LIN {X -0.019,Y -439.634,Z 747.550,A 0.000,B 0.000,C 90.000,E1 134.960} C_DIS
LIN {X -0.236,Y -446.877,Z 747.546,A 0.000,B 0.000,C 90.000,E1 134.271} C_DIS
LIN {X -0.116,Y -458.331,Z 747.539,A 0.000,B 0.000,C 90.000,E1 133.095} C_DIS
LIN {X 0.017,Y -466.662,Z 747.535,A 0.000,B 0.000,C 90.000,E1 132.204} C_DIS
LIN {X 0.112,Y -474.907,Z 747.530,A 0.000,B 0.000,C 90.000,E1 131.310} C_DIS
LIN {X -0.249,Y -482.897,Z 747.525,A 0.000,B 0.000,C 90.000,E1 130.458} C_DIS
LIN {X 0.218,Y -489.352,Z 747.520,A 0.000,B 0.000,C 90.000,E1 129.644} C_DIS
LIN {X 0.055,Y -494.191,Z 747.517,A 0.000,B 0.000,C 90.000,E1 129.072} C_DIS
LIN {X 0.218,Y -496.646,Z 747.515,A 0.000,B 0.000,C 90.000,E1 128.749} C_DIS
LIN {X -0.083,Y -504.313,Z 747.510,A 0.000,B 0.000,C 90.000,E1 127.729} C_DIS
LIN {X 0.206,Y -509.388,Z 747.505,A 0.000,B 0.000,C 90.000,E1 126.950} C_DIS
LIN {X 0.138,Y -513.980,Z 747.501,A 0.000,B 0.000,C 90.000,E1 126.217} C_DIS
LIN {X 0.118,Y -517.480,Z 747.498,A 0.000,B 0.000,C 90.000,E1 125.644} C_DIS
LIN {X -0.310,Y -520.857,Z 747.495,A 0.000,B 0.000,C 90.000,E1 125.105} C_DIS
LIN {X 0.174,Y -526.566,Z 747.489,A 0.000,B 0.000,C 90.000,E1 123.913} C_DIS
LIN {X -0.212,Y -530.567,Z 747.484,A 0.000,B 0.000,C 90.000,E1 123.086} C_DIS
LIN {X 0.022,Y -535.010,Z 747.478,A 0.000,B 0.000,C 90.000,E1 122.054} C_DIS
LIN {X -0.107,Y -538.597,Z 747.473,A 0.000,B 0.000,C 90.000,E1 121.209} C_DIS
LIN {X 0.079,Y -541.957,Z 747.469,A 0.000,B 0.000,C 90.000,E1 120.335} C_DIS
LIN {X -0.181,Y -544.080,Z 747.465,A 0.000,B 0.000,C 90.000,E1 119.795} C_DIS
LIN {X -0.209,Y -547.156,Z 747.461,A 0.000,B 0.000,C 90.000,E1 118.949} C_DIS
LIN {X -0.201,Y -550.028,Z 747.456,A 0.000,B 0.000,C 90.000,E1 118.103} C_DIS
LIN {X -0.163,Y -552.767,Z 747.451,A 0.000,B 0.000,C 90.000,E1 117.257} C_DIS
LIN {X -0.099,Y -555.288,Z 747.447,A 0.000,B 0.000,C 90.000,E1 116.411} C_DIS
LIN {X -0.256,Y -557.387,Z 747.442,A 0.000,B 0.000,C 90.000,E1 115.591} C_DIS
LIN {X 0.120,Y -559.196,Z 747.437,A 0.000,B 0.000,C 90.000,E1 114.719} C_DIS
LIN {X -0.194,Y -561.181,Z 747.431,A 0.000,B 0.000,C 90.000,E1 113.643} C_DIS
LIN {X 0.028,Y -562.877,Z 747.425,A 0.000,B 0.000,C 90.000,E1 112.514} C_DIS
LIN {X -0.020,Y -565.156,Z 747.416,A 0.000,B 0.000,C 90.000,E1 110.865} C_DIS
LIN {X 0.045,Y -566.668,Z 747.410,A 0.000,B 0.000,C 90.000,E1 109.758} C_DIS
LIN {X -0.105,Y -568.686,Z 747.401,A 0.000,B 0.000,C 90.000,E1 108.127} C_DIS
LIN {X -0.220,Y -570.542,Z 747.392,A 0.000,B 0.000,C 90.000,E1 106.496} C_DIS
LIN {X 0.268,Y -572.608,Z 747.381,A 0.000,B 0.000,C 90.000,E1 104.537} C_DIS
LIN {X -0.093,Y -574.375,Z 747.372,A 0.000,B 0.000,C 90.000,E1 102.939} C_DIS
LIN {X -0.200,Y -575.877,Z 747.364,A 0.000,B 0.000,C 90.000,E1 101.591} C_DIS
LIN {X -0.178,Y -577.585,Z 747.355,A 0.000,B 0.000,C 90.000,E1 99.962} C_DIS
LIN {X 0.234,Y -578.955,Z 747.348,A 0.000,B 0.000,C 90.000,E1 98.568} C_DIS
LIN {X -0.199,Y -580.736,Z 747.337,A 0.000,B 0.000,C 90.000,E1 96.720} C_DIS
LIN {X 0.183,Y -581.859,Z 747.330,A 0.000,B 0.000,C 90.000,E1 95.334} C_DIS
LIN {X -0.057,Y -582.888,Z 747.322,A 0.000,B 0.000,C 90.000,E1 94.012} C_DIS
LIN {X -0.138,Y -584.060,Z 747.313,A 0.000,B 0.000,C 90.000,E1 92.407} C_DIS
LIN {X 0.026,Y -584.828,Z 747.307,A 0.000,B 0.000,C 90.000,E1 91.318} C_DIS
LIN {X 0.164,Y -585.782,Z 747.297,A 0.000,B 0.000,C 90.000,E1 89.427} C_DIS
LIN {X 0.146,Y -586.397,Z 747.288,A 0.000,B 0.000,C 90.000,E1 87.822} C_DIS
LIN {X 0.139,Y -586.904,Z 747.279,A 0.000,B 0.000,C 90.000,E1 86.216} C_DIS
LIN {X -0.197,Y -587.126,Z 747.273,A 0.000,B 0.000,C 90.000,E1 85.179} C_DIS
LIN {X -0.163,Y -587.343,Z 747.264,A 0.000,B 0.000,C 90.000,E1 83.571} C_DIS
LIN {X -0.247,Y -587.387,Z 747.257,A 0.000,B 0.000,C 90.000,E1 82.243} C_DIS
LIN {X -0.084,Y -587.316,Z 747.248,A 0.000,B 0.000,C 90.000,E1 80.622} C_DIS
LIN {X -0.083,Y -587.056,Z 747.240,A 0.000,B 0.000,C 90.000,E1 79.285} C_DIS
LIN {X 0.276,Y -586.543,Z 747.232,A 0.000,B 0.000,C 90.000,E1 77.645} C_DIS
LIN {X -0.195,Y -586.012,Z 747.224,A 0.000,B 0.000,C 90.000,E1 76.353} C_DIS
LIN {X -0.292,Y -585.221,Z 747.215,A 0.000,B 0.000,C 90.000,E1 74.755} C_DIS
LIN {X 0.082,Y -584.442,Z 747.208,A 0.000,B 0.000,C 90.000,E1 73.378} C_DIS
LIN {X 0.044,Y -583.756,Z 747.202,A 0.000,B 0.000,C 90.000,E1 72.308} C_DIS
LIN {X 0.228,Y -582.538,Z 747.193,A 0.000,B 0.000,C 90.000,E1 70.678} C_DIS
LIN {X -0.015,Y -581.674,Z 747.187,A 0.000,B 0.000,C 90.000,E1 69.625} C_DIS
LIN {X -0.071,Y -580.407,Z 747.179,A 0.000,B 0.000,C 90.000,E1 68.284} C_DIS
LIN {X 0.057,Y -578.988,Z 747.172,A 0.000,B 0.000,C 90.000,E1 66.922} C_DIS
LIN {X -0.374,Y -577.316,Z 747.164,A 0.000,B 0.000,C 90.000,E1 65.613} C_DIS
LIN {X 0.172,Y -575.385,Z 747.157,A 0.000,B 0.000,C 90.000,E1 64.204} C_DIS
LIN {X 0.074,Y -573.609,Z 747.151,A 0.000,B 0.000,C 90.000,E1 63.127} C_DIS
LIN {X 0.103,Y -572.094,Z 747.146,A 0.000,B 0.000,C 90.000,E1 62.308} C_DIS
LIN {X 0.043,Y -571.055,Z 747.143,A 0.000,B 0.000,C 90.000,E1 61.769} C_DIS
LIN {X 0.136,Y -568.559,Z 747.137,A 0.000,B 0.000,C 90.000,E1 60.667} C_DIS
LIN {X -0.120,Y -566.513,Z 747.133,A 0.000,B 0.000,C 90.000,E1 59.871} C_DIS
LIN {X 0.184,Y -563.488,Z 747.127,A 0.000,B 0.000,C 90.000,E1 58.742} C_DIS
LIN {X 0.172,Y -560.988,Z 747.122,A 0.000,B 0.000,C 90.000,E1 57.916} C_DIS
LIN {X -0.164,Y -558.261,Z 747.117,A 0.000,B 0.000,C 90.000,E1 57.120} C_DIS
LIN {X -0.152,Y -554.192,Z 747.111,A 0.000,B 0.000,C 90.000,E1 56.008} C_DIS
LIN {X -0.067,Y -550.147,Z 747.106,A 0.000,B 0.000,C 90.000,E1 55.022} C_DIS
LIN {X -0.086,Y -546.928,Z 747.102,A 0.000,B 0.000,C 90.000,E1 54.322} C_DIS
LIN {X -0.279,Y -542.565,Z 747.097,A 0.000,B 0.000,C 90.000,E1 53.497} C_DIS
LIN {X -0.072,Y -540.308,Z 747.095,A 0.000,B 0.000,C 90.000,E1 53.050} C_DIS
LIN {X -0.187,Y -536.083,Z 747.091,A 0.000,B 0.000,C 90.000,E1 52.351} C_DIS
LIN {X 0.152,Y -532.406,Z 747.088,A 0.000,B 0.000,C 90.000,E1 51.743} C_DIS
LIN {X 0.133,Y -528.356,Z 747.084,A 0.000,B 0.000,C 90.000,E1 51.170} C_DIS
LIN {X 0.082,Y -523.734,Z 747.081,A 0.000,B 0.000,C 90.000,E1 50.598} C_DIS
LIN {X -0.207,Y -519.937,Z 747.079,A 0.000,B 0.000,C 90.000,E1 50.194} C_DIS
LIN {X -0.127,Y -514.436,Z 747.076,A 0.000,B 0.000,C 90.000,E1 49.622} C_DIS
LIN {X -0.008,Y -508.929,Z 747.073,A 0.000,B 0.000,C 90.000,E1 49.094} C_DIS
LIN {X 0.013,Y -504.675,Z 747.071,A 0.000,B 0.000,C 90.000,E1 48.728} C_DIS
LIN {X -0.184,Y -497.064,Z 747.068,A 0.000,B 0.000,C 90.000,E1 48.162} C_DIS
LIN {X 0.042,Y -490.703,Z 747.065,A 0.000,B 0.000,C 90.000,E1 47.676} C_DIS
LIN {X 0.313,Y -485.892,Z 747.063,A 0.000,B 0.000,C 90.000,E1 47.310} C_DIS
LIN {X 0.124,Y -479.241,Z 747.061,A 0.000,B 0.000,C 90.000,E1 46.905} C_DIS
LIN {X 0.132,Y -464.679,Z 747.056,A 0.000,B 0.000,C 90.000,E1 45.972} C_DIS
LIN {X -0.056,Y -446.780,Z 747.049,A 0.000,B 0.000,C 90.000,E1 44.838} C_DIS
LIN {X -0.086,Y -424.493,Z 747.041,A 0.000,B 0.000,C 90.000,E1 43.299} C_DIS
LIN {X -0.037,Y -418.213,Z 747.038,A 0.000,B 0.000,C 90.000,E1 42.813} C_DIS
LIN {X 0.002,Y -413.026,Z 747.035,A 0.000,B 0.000,C 90.000,E1 42.366} C_DIS
LIN {X -0.027,Y -412.987,Z 747.035,A 0.000,B 0.000,C 90.000,E1 42.366} C_DIS
LIN {X -0.059,Y -405.949,Z 747.014,A 0.000,B 0.000,C 90.000,E1 38.543} C_DIS
LIN {X 0.058,Y -402.213,Z 747.004,A 0.000,B 0.000,C 90.000,E1 36.790} C_DIS
LIN {X -0.041,Y -401.945,Z 747.004,A 0.000,B 0.000,C 90.000,E1 36.629} C_DIS
LIN {X -0.022,Y -402.376,Z 746.987,A 0.000,B 0.000,C 90.000,E1 33.658} C_DIS
LIN {X -0.078,Y -403.741,Z 746.968,A 0.000,B 0.000,C 90.000,E1 30.178} C_DIS
LIN {X -0.117,Y -405.368,Z 746.950,A 0.000,B 0.000,C 90.000,E1 27.052} C_DIS
LIN {X 0.102,Y -406.865,Z 746.937,A 0.000,B 0.000,C 90.000,E1 24.591} C_DIS
LIN {X -0.051,Y -409.155,Z 746.921,A 0.000,B 0.000,C 90.000,E1 21.844} C_DIS
LIN {X -0.182,Y -412.799,Z 746.902,A 0.000,B 0.000,C 90.000,E1 18.417} C_DIS
LIN {X 0.068,Y -416.776,Z 746.885,A 0.000,B 0.000,C 90.000,E1 15.300} C_DIS
LIN {X -0.087,Y -420.303,Z 746.872,A 0.000,B 0.000,C 90.000,E1 12.939} C_DIS
LIN {X 0.010,Y -423.521,Z 746.861,A 0.000,B 0.000,C 90.000,E1 10.894} C_DIS
LIN {X 0.205,Y -427.248,Z 746.847,A 0.000,B 0.000,C 90.000,E1 8.511} C_DIS
LIN {X -0.099,Y -430.434,Z 746.836,A 0.000,B 0.000,C 90.000,E1 6.543} C_DIS
LIN {X 0.080,Y -434.348,Z 746.823,A 0.000,B 0.000,C 90.000,E1 4.188} C_DIS
LIN {X -0.182,Y -437.889,Z 746.812,A 0.000,B 0.000,C 90.000,E1 2.236} C_DIS
LIN {X 0.056,Y -441.622,Z 746.801,A 0.000,B 0.000,C 90.000,E1 0.229} C_DIS
LIN {X 0.214,Y -447.043,Z 746.786,A 0.000,B 0.000,C 90.000,E1 357.478} C_DIS
LIN {X 0.098,Y -450.544,Z 746.777,A 0.000,B 0.000,C 90.000,E1 355.869} C_DIS
LIN {X -0.037,Y -455.589,Z 746.765,A 0.000,B 0.000,C 90.000,E1 353.628} C_DIS
LIN {X 0.107,Y -459.211,Z 746.756,A 0.000,B 0.000,C 90.000,E1 352.008} C_DIS
LIN {X 0.078,Y -461.979,Z 746.749,A 0.000,B 0.000,C 90.000,E1 350.735} C_DIS
LIN {X 0.166,Y -464.555,Z 746.742,A 0.000,B 0.000,C 90.000,E1 349.454} C_DIS
LIN {X -0.165,Y -466.988,Z 746.735,A 0.000,B 0.000,C 90.000,E1 348.229} C_DIS
LIN {X 0.182,Y -470.463,Z 746.724,A 0.000,B 0.000,C 90.000,E1 346.297} C_DIS
LIN {X 0.206,Y -474.757,Z 746.712,A 0.000,B 0.000,C 90.000,E1 344.102} C_DIS
LIN {X -0.042,Y -477.258,Z 746.707,A 0.000,B 0.000,C 90.000,E1 343.196} C_DIS
LIN {X 0.004,Y -478.941,Z 746.704,A 0.000,B 0.000,C 90.000,E1 342.725} C_DIS
LIN {X 0.105,Y -481.450,Z 746.701,A 0.000,B 0.000,C 90.000,E1 342.181} C_DIS
LIN {X -0.290,Y -484.359,Z 746.699,A 0.000,B 0.000,C 90.000,E1 341.764} C_DIS
LIN {X -0.218,Y -487.184,Z 746.697,A 0.000,B 0.000,C 90.000,E1 341.402} C_DIS
LIN {X 0.207,Y -493.459,Z 746.693,A 0.000,B 0.000,C 90.000,E1 340.732} C_DIS
LIN {X 0.081,Y -497.451,Z 746.691,A 0.000,B 0.000,C 90.000,E1 340.423} C_DIS
LIN {X 0.104,Y -506.768,Z 746.688,A 0.000,B 0.000,C 90.000,E1 339.752} C_DIS
LIN {X 0.237,Y -519.655,Z 746.683,A 0.000,B 0.000,C 90.000,E1 338.901} C_DIS
LIN {X 0.165,Y -534.050,Z 746.678,A 0.000,B 0.000,C 90.000,E1 338.050} C_DIS
LIN {X 0.076,Y -540.240,Z 746.676,A 0.000,B 0.000,C 90.000,E1 337.667} C_DIS
LIN {X 0.279,Y -546.445,Z 746.674,A 0.000,B 0.000,C 90.000,E1 337.230} C_DIS
LIN {X 0.259,Y -552.182,Z 746.671,A 0.000,B 0.000,C 90.000,E1 336.794} C_DIS
LIN {X -0.110,Y -557.650,Z 746.669,A 0.000,B 0.000,C 90.000,E1 336.357} C_DIS
LIN {X 0.016,Y -562.783,Z 746.666,A 0.000,B 0.000,C 90.000,E1 335.845} C_DIS
LIN {X 0.110,Y -567.837,Z 746.663,A 0.000,B 0.000,C 90.000,E1 335.305} C_DIS
LIN {X 0.126,Y -575.159,Z 746.658,A 0.000,B 0.000,C 90.000,E1 334.485} C_DIS
LIN {X -0.003,Y -580.902,Z 746.655,A 0.000,B 0.000,C 90.000,E1 333.819} C_DIS
LIN {X 0.186,Y -586.316,Z 746.651,A 0.000,B 0.000,C 90.000,E1 333.127} C_DIS
LIN {X -0.261,Y -594.686,Z 746.645,A 0.000,B 0.000,C 90.000,E1 332.103} C_DIS
LIN {X -0.322,Y -602.531,Z 746.639,A 0.000,B 0.000,C 90.000,E1 331.051} C_DIS
LIN {X -0.274,Y -609.960,Z 746.633,A 0.000,B 0.000,C 90.000,E1 329.999} C_DIS
LIN {X -0.127,Y -616.913,Z 746.628,A 0.000,B 0.000,C 90.000,E1 328.948} C_DIS
LIN {X -0.093,Y -623.424,Z 746.622,A 0.000,B 0.000,C 90.000,E1 327.916} C_DIS
LIN {X -0.302,Y -629.508,Z 746.616,A 0.000,B 0.000,C 90.000,E1 326.914} C_DIS
LIN {X -0.107,Y -633.737,Z 746.612,A 0.000,B 0.000,C 90.000,E1 326.135} C_DIS
LIN {X -0.209,Y -638.553,Z 746.607,A 0.000,B 0.000,C 90.000,E1 325.261} C_DIS
LIN {X 0.085,Y -642.410,Z 746.603,A 0.000,B 0.000,C 90.000,E1 324.482} C_DIS
LIN {X 0.343,Y -647.843,Z 746.597,A 0.000,B 0.000,C 90.000,E1 323.336} C_DIS
LIN {X -0.178,Y -651.259,Z 746.592,A 0.000,B 0.000,C 90.000,E1 322.637} C_DIS
LIN {X -0.277,Y -654.513,Z 746.588,A 0.000,B 0.000,C 90.000,E1 321.904} C_DIS
LIN {X 0.122,Y -658.536,Z 746.583,A 0.000,B 0.000,C 90.000,E1 320.884} C_DIS
LIN {X 0.095,Y -661.400,Z 746.579,A 0.000,B 0.000,C 90.000,E1 320.150} C_DIS
LIN {X 0.071,Y -665.025,Z 746.573,A 0.000,B 0.000,C 90.000,E1 319.175} C_DIS
LIN {X -0.406,Y -668.422,Z 746.568,A 0.000,B 0.000,C 90.000,E1 318.243} C_DIS
LIN {X 0.109,Y -671.560,Z 746.563,A 0.000,B 0.000,C 90.000,E1 317.229} C_DIS
LIN {X -0.262,Y -675.224,Z 746.556,A 0.000,B 0.000,C 90.000,E1 316.053} C_DIS
LIN {X -0.142,Y -677.964,Z 746.550,A 0.000,B 0.000,C 90.000,E1 315.081} C_DIS
LIN {X -0.028,Y -679.852,Z 746.546,A 0.000,B 0.000,C 90.000,E1 314.352} C_DIS
LIN {X -0.219,Y -683.274,Z 746.538,A 0.000,B 0.000,C 90.000,E1 312.933} C_DIS
LIN {X -0.008,Y -685.425,Z 746.533,A 0.000,B 0.000,C 90.000,E1 311.962} C_DIS
LIN {X -0.050,Y -688.297,Z 746.525,A 0.000,B 0.000,C 90.000,E1 310.539} C_DIS
LIN {X 0.281,Y -689.855,Z 746.520,A 0.000,B 0.000,C 90.000,E1 309.564} C_DIS
LIN {X 0.196,Y -691.217,Z 746.515,A 0.000,B 0.000,C 90.000,E1 308.624} C_DIS
LIN {X 0.196,Y -692.765,Z 746.508,A 0.000,B 0.000,C 90.000,E1 307.443} C_DIS
LIN {X -0.208,Y -694.053,Z 746.502,A 0.000,B 0.000,C 90.000,E1 306.297} C_DIS
LIN {X -0.030,Y -695.135,Z 746.495,A 0.000,B 0.000,C 90.000,E1 305.105} C_DIS
LIN {X 0.164,Y -696.072,Z 746.489,A 0.000,B 0.000,C 90.000,E1 303.913} C_DIS
LIN {X -0.117,Y -697.374,Z 746.479,A 0.000,B 0.000,C 90.000,E1 302.291} C_DIS
LIN {X -0.022,Y -698.460,Z 746.472,A 0.000,B 0.000,C 90.000,E1 300.875} C_DIS
LIN {X -0.097,Y -698.842,Z 746.468,A 0.000,B 0.000,C 90.000,E1 300.178} C_DIS
LIN {X -0.004,Y -699.217,Z 746.461,A 0.000,B 0.000,C 90.000,E1 298.999} C_DIS
LIN {X -0.313,Y -699.741,Z 746.452,A 0.000,B 0.000,C 90.000,E1 297.385} C_DIS
LIN {X -0.372,Y -700.665,Z 746.440,A 0.000,B 0.000,C 90.000,E1 295.283} C_DIS
LIN {X 0.174,Y -700.699,Z 746.438,A 0.000,B 0.000,C 90.000,E1 294.771} C_DIS
LIN {X -0.191,Y -700.580,Z 746.436,A 0.000,B 0.000,C 90.000,E1 294.567} C_DIS
LIN {X 0.061,Y -699.745,Z 746.434,A 0.000,B 0.000,C 90.000,E1 294.079} C_DIS
LIN {X 0.329,Y -698.958,Z 746.433,A 0.000,B 0.000,C 90.000,E1 293.823} C_DIS
LIN {X -0.326,Y -697.585,Z 746.431,A 0.000,B 0.000,C 90.000,E1 293.643} C_DIS
LIN {X 0.062,Y -695.117,Z 746.429,A 0.000,B 0.000,C 90.000,E1 293.259} C_DIS
LIN {X 0.187,Y -693.835,Z 746.429,A 0.000,B 0.000,C 90.000,E1 293.131} C_DIS
LIN {X 0.094,Y -691.936,Z 746.428,A 0.000,B 0.000,C 90.000,E1 293.025} C_DIS
LIN {X -0.145,Y -686.391,Z 746.426,A 0.000,B 0.000,C 90.000,E1 292.770} C_DIS
LIN {X -0.164,Y -684.592,Z 746.426,A 0.000,B 0.000,C 90.000,E1 292.695} C_DIS
LIN {X 0.082,Y -676.168,Z 746.425,A 0.000,B 0.000,C 90.000,E1 292.461} C_DIS
LIN {X 0.077,Y -667.423,Z 746.424,A 0.000,B 0.000,C 90.000,E1 292.333} C_DIS
LIN {X -0.087,Y -661.307,Z 746.424,A 0.000,B 0.000,C 90.000,E1 292.280} C_DIS
LIN {X 0.009,Y -647.994,Z 746.423,A 0.000,B 0.000,C 90.000,E1 292.078} C_DIS
LIN {X 0.020,Y -638.305,Z 746.422,A 0.000,B 0.000,C 90.000,E1 291.897} C_DIS
LIN {X 0.148,Y -624.929,Z 746.420,A 0.000,B 0.000,C 90.000,E1 291.589} C_DIS
LIN {X 0.204,Y -607.988,Z 746.418,A 0.000,B 0.000,C 90.000,E1 291.153} C_DIS
LIN {X -0.258,Y -574.712,Z 746.412,A 0.000,B 0.000,C 90.000,E1 290.248} C_DIS
LIN {X -0.157,Y -567.276,Z 746.411,A 0.000,B 0.000,C 90.000,E1 290.047} C_DIS
LIN {X -0.165,Y -562.140,Z 746.410,A 0.000,B 0.000,C 90.000,E1 289.866} C_DIS
LIN {X -0.244,Y -560.675,Z 746.410,A 0.000,B 0.000,C 90.000,E1 289.812} C_DIS
LIN {X 0.015,Y -556.891,Z 746.409,A 0.000,B 0.000,C 90.000,E1 289.577} C_DIS
LIN {X 0.243,Y -555.751,Z 746.408,A 0.000,B 0.000,C 90.000,E1 289.396} C_DIS
LIN {X 0.197,Y -555.730,Z 746.408,A 0.000,B 0.000,C 90.000,E1 289.396} C_DIS
LIN {X 0.164,Y -555.085,Z 746.406,A 0.000,B 0.000,C 90.000,E1 289.087} C_DIS
LIN {X 0.313,Y -554.658,Z 746.402,A 0.000,B 0.000,C 90.000,E1 288.236} C_DIS
LIN {X -0.272,Y -554.104,Z 746.392,A 0.000,B 0.000,C 90.000,E1 286.622} C_DIS
LIN {X 0.203,Y -553.457,Z 746.383,A 0.000,B 0.000,C 90.000,E1 284.898} C_DIS
LIN {X 0.236,Y -552.788,Z 746.372,A 0.000,B 0.000,C 90.000,E1 282.939} C_DIS
LIN {X -0.129,Y -552.233,Z 746.363,A 0.000,B 0.000,C 90.000,E1 281.299} C_DIS
LIN {X -0.182,Y -551.764,Z 746.355,A 0.000,B 0.000,C 90.000,E1 279.905} C_DIS
LIN {X -0.240,Y -551.110,Z 746.347,A 0.000,B 0.000,C 90.000,E1 278.511} C_DIS
LIN {X 0.265,Y -550.342,Z 746.338,A 0.000,B 0.000,C 90.000,E1 276.777} C_DIS
LIN {X 0.140,Y -549.539,Z 746.328,A 0.000,B 0.000,C 90.000,E1 275.106} C_DIS
LIN {X 0.075,Y -548.340,Z 746.316,A 0.000,B 0.000,C 90.000,E1 272.865} C_DIS
LIN {X -0.125,Y -547.324,Z 746.305,A 0.000,B 0.000,C 90.000,E1 270.917} C_DIS
LIN {X 0.058,Y -546.647,Z 746.299,A 0.000,B 0.000,C 90.000,E1 269.771} C_DIS
LIN {X -0.220,Y -545.502,Z 746.289,A 0.000,B 0.000,C 90.000,E1 268.108} C_DIS
LIN {X 0.023,Y -544.459,Z 746.280,A 0.000,B 0.000,C 90.000,E1 266.388} C_DIS
LIN {X 0.244,Y -543.555,Z 746.272,A 0.000,B 0.000,C 90.000,E1 264.951} C_DIS
LIN {X -0.024,Y -542.371,Z 746.263,A 0.000,B 0.000,C 90.000,E1 263.280} C_DIS
LIN {X 0.282,Y -540.984,Z 746.253,A 0.000,B 0.000,C 90.000,E1 261.546} C_DIS
LIN {X 0.108,Y -539.572,Z 746.244,A 0.000,B 0.000,C 90.000,E1 259.859} C_DIS
LIN {X -0.102,Y -538.169,Z 746.234,A 0.000,B 0.000,C 90.000,E1 258.173} C_DIS
LIN {X 0.092,Y -537.493,Z 746.230,A 0.000,B 0.000,C 90.000,E1 257.297} C_DIS
LIN {X -0.007,Y -536.191,Z 746.222,A 0.000,B 0.000,C 90.000,E1 255.880} C_DIS
LIN {X -0.177,Y -534.950,Z 746.215,A 0.000,B 0.000,C 90.000,E1 254.755} C_DIS
LIN {X -0.178,Y -533.372,Z 746.207,A 0.000,B 0.000,C 90.000,E1 253.323} C_DIS
LIN {X -0.023,Y -531.514,Z 746.198,A 0.000,B 0.000,C 90.000,E1 251.583} C_DIS
LIN {X -0.318,Y -530.904,Z 746.195,A 0.000,B 0.000,C 90.000,E1 251.040} C_DIS
LIN {X 0.125,Y -528.550,Z 746.185,A 0.000,B 0.000,C 90.000,E1 249.263} C_DIS
LIN {X -0.149,Y -526.543,Z 746.177,A 0.000,B 0.000,C 90.000,E1 247.847} C_DIS
LIN {X -0.090,Y -523.902,Z 746.167,A 0.000,B 0.000,C 90.000,E1 246.102} C_DIS
LIN {X 0.070,Y -522.028,Z 746.161,A 0.000,B 0.000,C 90.000,E1 244.921} C_DIS
LIN {X -0.053,Y -520.139,Z 746.154,A 0.000,B 0.000,C 90.000,E1 243.768} C_DIS
LIN {X 0.130,Y -518.626,Z 746.149,A 0.000,B 0.000,C 90.000,E1 242.871} C_DIS
LIN {X -0.043,Y -516.421,Z 746.143,A 0.000,B 0.000,C 90.000,E1 241.719} C_DIS
LIN {X -0.002,Y -512.994,Z 746.133,A 0.000,B 0.000,C 90.000,E1 239.950} C_DIS
LIN {X 0.144,Y -510.107,Z 746.125,A 0.000,B 0.000,C 90.000,E1 238.456} C_DIS
LIN {X 0.018,Y -508.337,Z 746.120,A 0.000,B 0.000,C 90.000,E1 237.582} C_DIS
LIN {X -0.130,Y -506.432,Z 746.115,A 0.000,B 0.000,C 90.000,E1 236.707} C_DIS
LIN {X 0.176,Y -503.141,Z 746.107,A 0.000,B 0.000,C 90.000,E1 235.182} C_DIS
LIN {X 0.128,Y -500.327,Z 746.100,A 0.000,B 0.000,C 90.000,E1 233.989} C_DIS
LIN {X -0.238,Y -498.091,Z 746.095,A 0.000,B 0.000,C 90.000,E1 233.130} C_DIS
LIN {X -0.179,Y -492.770,Z 746.083,A 0.000,B 0.000,C 90.000,E1 231.009} C_DIS
LIN {X -0.120,Y -487.009,Z 746.070,A 0.000,B 0.000,C 90.000,E1 228.566} C_DIS
LIN {X -0.049,Y -483.635,Z 746.061,A 0.000,B 0.000,C 90.000,E1 227.025} C_DIS
LIN {X 0.068,Y -479.669,Z 746.051,A 0.000,B 0.000,C 90.000,E1 225.162} C_DIS
LIN {X -0.013,Y -476.391,Z 746.042,A 0.000,B 0.000,C 90.000,E1 223.623} C_DIS
LIN {X -0.017,Y -474.386,Z 746.037,A 0.000,B 0.000,C 90.000,E1 222.690} C_DIS
LIN {X 0.048,Y -471.689,Z 746.030,A 0.000,B 0.000,C 90.000,E1 221.434} C_DIS
LIN {X -0.050,Y -467.496,Z 746.020,A 0.000,B 0.000,C 90.000,E1 219.564} C_DIS
LIN {X -0.127,Y -462.737,Z 746.008,A 0.000,B 0.000,C 90.000,E1 217.363} C_DIS
LIN {X -0.137,Y -457.474,Z 745.993,A 0.000,B 0.000,C 90.000,E1 214.818} C_DIS
LIN {X -0.009,Y -453.640,Z 745.983,A 0.000,B 0.000,C 90.000,E1 212.880} C_DIS
LIN {X 0.076,Y -450.655,Z 745.974,A 0.000,B 0.000,C 90.000,E1 211.258} C_DIS
LIN {X -0.127,Y -447.615,Z 745.965,A 0.000,B 0.000,C 90.000,E1 209.667} C_DIS
LIN {X -0.131,Y -445.844,Z 745.959,A 0.000,B 0.000,C 90.000,E1 208.693} C_DIS
LIN {X -0.193,Y -442.224,Z 745.948,A 0.000,B 0.000,C 90.000,E1 206.744} C_DIS
LIN {X -0.022,Y -439.774,Z 745.941,A 0.000,B 0.000,C 90.000,E1 205.412} C_DIS
LIN {X -0.054,Y -436.692,Z 745.932,A 0.000,B 0.000,C 90.000,E1 203.770} C_DIS
LIN {X 0.068,Y -432.993,Z 745.921,A 0.000,B 0.000,C 90.000,E1 201.770} C_DIS
LIN {X 0.198,Y -427.956,Z 745.906,A 0.000,B 0.000,C 90.000,E1 199.087} C_DIS
LIN {X 0.069,Y -425.492,Z 745.899,A 0.000,B 0.000,C 90.000,E1 197.764} C_DIS
LIN {X -0.080,Y -420.869,Z 745.886,A 0.000,B 0.000,C 90.000,E1 195.426} C_DIS
LIN {X -0.176,Y -416.465,Z 745.872,A 0.000,B 0.000,C 90.000,E1 193.063} C_DIS
LIN {X 0.113,Y -414.067,Z 745.865,A 0.000,B 0.000,C 90.000,E1 191.658} C_DIS
LIN {X 0.056,Y -409.923,Z 745.852,A 0.000,B 0.000,C 90.000,E1 189.265} C_DIS
LIN {X 0.147,Y -405.915,Z 745.838,A 0.000,B 0.000,C 90.000,E1 186.834} C_DIS
LIN {X 0.082,Y -403.209,Z 745.828,A 0.000,B 0.000,C 90.000,E1 185.106} C_DIS
LIN {X -0.092,Y -400.207,Z 745.817,A 0.000,B 0.000,C 90.000,E1 183.037} C_DIS
LIN {X 0.074,Y -397.827,Z 745.807,A 0.000,B 0.000,C 90.000,E1 181.260} C_DIS
LIN {X -0.060,Y -394.231,Z 745.789,A 0.000,B 0.000,C 90.000,E1 178.108} C_DIS
LIN {X 0.049,Y -390.719,Z 745.770,A 0.000,B 0.000,C 90.000,E1 174.546} C_DIS
LIN {X -0.060,Y -387.885,Z 745.744,A 0.000,B 0.000,C 90.000,E1 169.926} C_DIS
LIN {X 0.022,Y -386.791,Z 745.730,A 0.000,B 0.000,C 90.000,E1 167.409} C_DIS
LIN {X -0.160,Y -386.073,Z 745.720,A 0.000,B 0.000,C 90.000,E1 165.644} C_DIS
LIN {X 0.166,Y -385.270,Z 745.704,A 0.000,B 0.000,C 90.000,E1 162.725} C_DIS
LIN {X -0.072,Y -384.754,Z 745.692,A 0.000,B 0.000,C 90.000,E1 160.604} C_DIS
LIN {X 0.168,Y -384.418,Z 745.680,A 0.000,B 0.000,C 90.000,E1 158.411} C_DIS
LIN {X -0.022,Y -384.134,Z 745.666,A 0.000,B 0.000,C 90.000,E1 155.921} C_DIS
LIN {X -0.122,Y -385.150,Z 745.636,A 0.000,B 0.000,C 90.000,E1 150.539} C_DIS
LIN {X 0.091,Y -386.726,Z 745.622,A 0.000,B 0.000,C 90.000,E1 147.995} C_DIS
LIN {X 0.018,Y -388.147,Z 745.612,A 0.000,B 0.000,C 90.000,E1 146.215} C_DIS
LIN {X 0.095,Y -392.492,Z 745.593,A 0.000,B 0.000,C 90.000,E1 142.637} C_DIS
LIN {X -0.124,Y -395.141,Z 745.585,A 0.000,B 0.000,C 90.000,E1 141.251} C_DIS
LIN {X -0.034,Y -395.938,Z 745.583,A 0.000,B 0.000,C 90.000,E1 140.884} C_DIS
LIN {X -0.149,Y -397.814,Z 745.579,A 0.000,B 0.000,C 90.000,E1 140.194} C_DIS
LIN {X -0.048,Y -399.150,Z 745.577,A 0.000,B 0.000,C 90.000,E1 139.828} C_DIS
LIN {X 0.060,Y -400.309,Z 745.575,A 0.000,B 0.000,C 90.000,E1 139.461} C_DIS
LIN {X 0.078,Y -402.798,Z 745.572,A 0.000,B 0.000,C 90.000,E1 138.933} C_DIS
LIN {X -0.115,Y -407.203,Z 745.568,A 0.000,B 0.000,C 90.000,E1 138.243} C_DIS
LIN {X -0.145,Y -410.376,Z 745.566,A 0.000,B 0.000,C 90.000,E1 137.838} C_DIS
LIN {X -0.120,Y -432.124,Z 745.553,A 0.000,B 0.000,C 90.000,E1 135.567} C_DIS
LIN {X -0.151,Y -445.370,Z 745.546,A 0.000,B 0.000,C 90.000,E1 134.271} C_DIS
LIN {X -0.102,Y -455.431,Z 745.540,A 0.000,B 0.000,C 90.000,E1 133.257} C_DIS
LIN {X -0.126,Y -461.026,Z 745.537,A 0.000,B 0.000,C 90.000,E1 132.690} C_DIS
LIN {X -0.117,Y -469.165,Z 745.532,A 0.000,B 0.000,C 90.000,E1 131.838} C_DIS
LIN {X 0.074,Y -474.634,Z 745.529,A 0.000,B 0.000,C 90.000,E1 131.229} C_DIS
LIN {X -0.105,Y -482.522,Z 745.524,A 0.000,B 0.000,C 90.000,E1 130.378} C_DIS
LIN {X -0.097,Y -488.860,Z 745.520,A 0.000,B 0.000,C 90.000,E1 129.644} C_DIS
LIN {X 0.075,Y -493.718,Z 745.517,A 0.000,B 0.000,C 90.000,E1 129.036} C_DIS
LIN {X 0.050,Y -496.126,Z 745.515,A 0.000,B 0.000,C 90.000,E1 128.749} C_DIS
LIN {X 0.035,Y -504.668,Z 745.509,A 0.000,B 0.000,C 90.000,E1 127.604} C_DIS
LIN {X -0.007,Y -509.640,Z 745.505,A 0.000,B 0.000,C 90.000,E1 126.870} C_DIS
LIN {X -0.187,Y -513.397,Z 745.502,A 0.000,B 0.000,C 90.000,E1 126.297} C_DIS
LIN {X 0.077,Y -517.038,Z 745.498,A 0.000,B 0.000,C 90.000,E1 125.678} C_DIS
LIN {X -0.050,Y -520.478,Z 745.495,A 0.000,B 0.000,C 90.000,E1 125.105} C_DIS
LIN {X 0.063,Y -525.659,Z 745.489,A 0.000,B 0.000,C 90.000,E1 124.072} C_DIS
LIN {X 0.153,Y -527.792,Z 745.487,A 0.000,B 0.000,C 90.000,E1 123.627} C_DIS
LIN {X 0.051,Y -533.639,Z 745.480,A 0.000,B 0.000,C 90.000,E1 122.339} C_DIS
LIN {X 0.045,Y -537.875,Z 745.474,A 0.000,B 0.000,C 90.000,E1 121.337} C_DIS
LIN {X 0.224,Y -541.288,Z 745.469,A 0.000,B 0.000,C 90.000,E1 120.463} C_DIS
LIN {X 0.178,Y -545.597,Z 745.463,A 0.000,B 0.000,C 90.000,E1 119.333} C_DIS
LIN {X -0.075,Y -549.543,Z 745.457,A 0.000,B 0.000,C 90.000,E1 118.231} C_DIS
LIN {X -0.041,Y -552.337,Z 745.452,A 0.000,B 0.000,C 90.000,E1 117.385} C_DIS
LIN {X 0.019,Y -554.921,Z 745.448,A 0.000,B 0.000,C 90.000,E1 116.539} C_DIS
LIN {X -0.142,Y -557.097,Z 745.443,A 0.000,B 0.000,C 90.000,E1 115.720} C_DIS
LIN {X -0.277,Y -558.993,Z 745.438,A 0.000,B 0.000,C 90.000,E1 114.899} C_DIS
LIN {X 0.120,Y -560.638,Z 745.434,A 0.000,B 0.000,C 90.000,E1 114.027} C_DIS
LIN {X -0.178,Y -562.419,Z 745.427,A 0.000,B 0.000,C 90.000,E1 112.950} C_DIS
LIN {X 0.170,Y -564.364,Z 745.420,A 0.000,B 0.000,C 90.000,E1 111.535} C_DIS
LIN {X 0.162,Y -566.664,Z 745.411,A 0.000,B 0.000,C 90.000,E1 109.885} C_DIS
LIN {X -0.141,Y -568.426,Z 745.403,A 0.000,B 0.000,C 90.000,E1 108.544} C_DIS
LIN {X -0.056,Y -569.992,Z 745.395,A 0.000,B 0.000,C 90.000,E1 107.166} C_DIS
LIN {X -0.121,Y -571.265,Z 745.389,A 0.000,B 0.000,C 90.000,E1 106.079} C_DIS
LIN {X -0.172,Y -573.342,Z 745.379,A 0.000,B 0.000,C 90.000,E1 104.175} C_DIS
LIN {X -0.297,Y -574.846,Z 745.371,A 0.000,B 0.000,C 90.000,E1 102.827} C_DIS
LIN {X 0.175,Y -576.360,Z 745.364,A 0.000,B 0.000,C 90.000,E1 101.422} C_DIS
LIN {X 0.218,Y -578.112,Z 745.355,A 0.000,B 0.000,C 90.000,E1 99.792} C_DIS
LIN {X -0.145,Y -579.212,Z 745.349,A 0.000,B 0.000,C 90.000,E1 98.746} C_DIS
LIN {X 0.084,Y -581.031,Z 745.338,A 0.000,B 0.000,C 90.000,E1 96.834} C_DIS
LIN {X 0.052,Y -582.404,Z 745.329,A 0.000,B 0.000,C 90.000,E1 95.220} C_DIS
LIN {X 0.192,Y -583.260,Z 745.323,A 0.000,B 0.000,C 90.000,E1 94.131} C_DIS
LIN {X 0.158,Y -584.461,Z 745.314,A 0.000,B 0.000,C 90.000,E1 92.522} C_DIS
LIN {X -0.072,Y -585.380,Z 745.307,A 0.000,B 0.000,C 90.000,E1 91.203} C_DIS
LIN {X -0.111,Y -586.221,Z 745.298,A 0.000,B 0.000,C 90.000,E1 89.599} C_DIS
LIN {X -0.119,Y -586.844,Z 745.289,A 0.000,B 0.000,C 90.000,E1 87.993} C_DIS
LIN {X -0.113,Y -587.369,Z 745.280,A 0.000,B 0.000,C 90.000,E1 86.388} C_DIS
LIN {X -0.254,Y -587.647,Z 745.273,A 0.000,B 0.000,C 90.000,E1 85.065} C_DIS
LIN {X -0.147,Y -587.833,Z 745.264,A 0.000,B 0.000,C 90.000,E1 83.451} C_DIS
LIN {X -0.292,Y -587.858,Z 745.256,A 0.000,B 0.000,C 90.000,E1 82.129} C_DIS
LIN {X -0.027,Y -587.789,Z 745.247,A 0.000,B 0.000,C 90.000,E1 80.500} C_DIS
LIN {X -0.010,Y -587.460,Z 745.240,A 0.000,B 0.000,C 90.000,E1 79.162} C_DIS
LIN {X -0.011,Y -587.012,Z 745.232,A 0.000,B 0.000,C 90.000,E1 77.825} C_DIS
LIN {X 0.230,Y -586.474,Z 745.225,A 0.000,B 0.000,C 90.000,E1 76.464} C_DIS
LIN {X -0.174,Y -585.521,Z 745.215,A 0.000,B 0.000,C 90.000,E1 74.629} C_DIS
LIN {X -0.117,Y -584.561,Z 745.206,A 0.000,B 0.000,C 90.000,E1 73.015} C_DIS
LIN {X 0.247,Y -583.565,Z 745.198,A 0.000,B 0.000,C 90.000,E1 71.638} C_DIS
LIN {X -0.119,Y -582.280,Z 745.189,A 0.000,B 0.000,C 90.000,E1 70.061} C_DIS
LIN {X -0.167,Y -581.044,Z 745.182,A 0.000,B 0.000,C 90.000,E1 68.720} C_DIS
LIN {X -0.029,Y -579.620,Z 745.174,A 0.000,B 0.000,C 90.000,E1 67.358} C_DIS
LIN {X -0.071,Y -578.367,Z 745.168,A 0.000,B 0.000,C 90.000,E1 66.282} C_DIS
LIN {X 0.013,Y -576.521,Z 745.161,A 0.000,B 0.000,C 90.000,E1 64.921} C_DIS
LIN {X -0.073,Y -574.840,Z 745.155,A 0.000,B 0.000,C 90.000,E1 63.845} C_DIS
LIN {X 0.073,Y -572.959,Z 745.149,A 0.000,B 0.000,C 90.000,E1 62.743} C_DIS
LIN {X 0.196,Y -570.771,Z 745.143,A 0.000,B 0.000,C 90.000,E1 61.641} C_DIS
LIN {X -0.038,Y -568.897,Z 745.138,A 0.000,B 0.000,C 90.000,E1 60.845} C_DIS
LIN {X 0.023,Y -566.078,Z 745.132,A 0.000,B 0.000,C 90.000,E1 59.744} C_DIS
LIN {X 0.032,Y -563.791,Z 745.127,A 0.000,B 0.000,C 90.000,E1 58.918} C_DIS
LIN {X 0.207,Y -561.309,Z 745.123,A 0.000,B 0.000,C 90.000,E1 58.074} C_DIS
LIN {X 0.172,Y -558.562,Z 745.118,A 0.000,B 0.000,C 90.000,E1 57.248} C_DIS
LIN {X -0.120,Y -554.461,Z 745.112,A 0.000,B 0.000,C 90.000,E1 56.167} C_DIS
LIN {X 0.087,Y -550.961,Z 745.107,A 0.000,B 0.000,C 90.000,E1 55.308} C_DIS
LIN {X 0.022,Y -549.068,Z 745.105,A 0.000,B 0.000,C 90.000,E1 54.895} C_DIS
LIN {X -0.009,Y -545.698,Z 745.101,A 0.000,B 0.000,C 90.000,E1 54.196} C_DIS
LIN {X 0.072,Y -542.791,Z 745.098,A 0.000,B 0.000,C 90.000,E1 53.623} C_DIS
LIN {X 0.132,Y -539.723,Z 745.095,A 0.000,B 0.000,C 90.000,E1 53.050} C_DIS
LIN {X 0.042,Y -535.398,Z 745.091,A 0.000,B 0.000,C 90.000,E1 52.351} C_DIS
LIN {X -0.256,Y -531.708,Z 745.088,A 0.000,B 0.000,C 90.000,E1 51.823} C_DIS
LIN {X -0.074,Y -527.733,Z 745.085,A 0.000,B 0.000,C 90.000,E1 51.251} C_DIS
LIN {X 0.203,Y -523.008,Z 745.082,A 0.000,B 0.000,C 90.000,E1 50.642} C_DIS
LIN {X 0.027,Y -519.190,Z 745.079,A 0.000,B 0.000,C 90.000,E1 50.231} C_DIS
LIN {X 0.134,Y -513.688,Z 745.076,A 0.000,B 0.000,C 90.000,E1 49.666} C_DIS
LIN {X -0.136,Y -507.975,Z 745.073,A 0.000,B 0.000,C 90.000,E1 49.175} C_DIS
LIN {X 0.139,Y -503.545,Z 745.071,A 0.000,B 0.000,C 90.000,E1 48.771} C_DIS
LIN {X 0.337,Y -495.748,Z 745.068,A 0.000,B 0.000,C 90.000,E1 48.162} C_DIS
LIN {X -0.084,Y -489.377,Z 745.065,A 0.000,B 0.000,C 90.000,E1 47.757} C_DIS
LIN {X 0.012,Y -482.877,Z 745.063,A 0.000,B 0.000,C 90.000,E1 47.310} C_DIS
LIN {X -0.175,Y -466.573,Z 745.057,A 0.000,B 0.000,C 90.000,E1 46.296} C_DIS
LIN {X 0.006,Y -448.629,Z 745.051,A 0.000,B 0.000,C 90.000,E1 45.121} C_DIS
LIN {X 0.122,Y -424.720,Z 745.042,A 0.000,B 0.000,C 90.000,E1 43.461} C_DIS
LIN {X 0.104,Y -415.835,Z 745.038,A 0.000,B 0.000,C 90.000,E1 42.771} C_DIS
LIN {X 0.198,Y -413.426,Z 745.036,A 0.000,B 0.000,C 90.000,E1 42.528} C_DIS
LIN {X 0.169,Y -413.390,Z 745.036,A 0.000,B 0.000,C 90.000,E1 42.528} C_DIS
LIN {X 0.071,Y -405.661,Z 745.013,A 0.000,B 0.000,C 90.000,E1 38.382} C_DIS
LIN {X 0.032,Y -402.275,Z 745.005,A 0.000,B 0.000,C 90.000,E1 36.824} C_DIS
LIN {X 0.095,Y -402.755,Z 744.986,A 0.000,B 0.000,C 90.000,E1 33.499} C_DIS
LIN {X -0.063,Y -404.026,Z 744.969,A 0.000,B 0.000,C 90.000,E1 30.384} C_DIS
LIN {X -0.086,Y -405.636,Z 744.951,A 0.000,B 0.000,C 90.000,E1 27.257} C_DIS
LIN {X -0.050,Y -407.108,Z 744.938,A 0.000,B 0.000,C 90.000,E1 24.823} C_DIS
LIN {X 0.168,Y -409.388,Z 744.923,A 0.000,B 0.000,C 90.000,E1 22.025} C_DIS
LIN {X 0.184,Y -413.357,Z 744.901,A 0.000,B 0.000,C 90.000,E1 18.236} C_DIS
LIN {X -0.057,Y -417.348,Z 744.884,A 0.000,B 0.000,C 90.000,E1 15.190} C_DIS
LIN {X 0.157,Y -420.359,Z 744.873,A 0.000,B 0.000,C 90.000,E1 13.119} C_DIS
LIN {X -0.154,Y -423.526,Z 744.862,A 0.000,B 0.000,C 90.000,E1 11.130} C_DIS
LIN {X -0.161,Y -425.612,Z 744.854,A 0.000,B 0.000,C 90.000,E1 9.782} C_DIS
LIN {X 0.143,Y -427.758,Z 744.847,A 0.000,B 0.000,C 90.000,E1 8.398} C_DIS
LIN {X 0.175,Y -430.414,Z 744.838,A 0.000,B 0.000,C 90.000,E1 6.720} C_DIS
LIN {X -0.033,Y -434.280,Z 744.825,A 0.000,B 0.000,C 90.000,E1 4.416} C_DIS
LIN {X -0.198,Y -438.373,Z 744.812,A 0.000,B 0.000,C 90.000,E1 2.121} C_DIS
LIN {X 0.051,Y -442.097,Z 744.801,A 0.000,B 0.000,C 90.000,E1 0.115} C_DIS
LIN {X 0.221,Y -447.281,Z 744.786,A 0.000,B 0.000,C 90.000,E1 357.478} C_DIS
LIN {X -0.188,Y -451.451,Z 744.775,A 0.000,B 0.000,C 90.000,E1 355.584} C_DIS
LIN {X -0.019,Y -455.793,Z 744.765,A 0.000,B 0.000,C 90.000,E1 353.628} C_DIS
LIN {X 0.129,Y -459.402,Z 744.756,A 0.000,B 0.000,C 90.000,E1 352.008} C_DIS
LIN {X 0.104,Y -462.169,Z 744.749,A 0.000,B 0.000,C 90.000,E1 350.735} C_DIS
LIN {X -0.005,Y -465.358,Z 744.740,A 0.000,B 0.000,C 90.000,E1 349.162} C_DIS
LIN {X 0.132,Y -467.713,Z 744.733,A 0.000,B 0.000,C 90.000,E1 347.881} C_DIS
LIN {X -0.240,Y -470.624,Z 744.724,A 0.000,B 0.000,C 90.000,E1 346.353} C_DIS
LIN {X 0.204,Y -475.504,Z 744.710,A 0.000,B 0.000,C 90.000,E1 343.795} C_DIS
LIN {X -0.002,Y -477.147,Z 744.707,A 0.000,B 0.000,C 90.000,E1 343.196} C_DIS
LIN {X -0.172,Y -478.080,Z 744.705,A 0.000,B 0.000,C 90.000,E1 342.906} C_DIS
LIN {X 0.020,Y -479.789,Z 744.702,A 0.000,B 0.000,C 90.000,E1 342.417} C_DIS
LIN {X 0.078,Y -482.014,Z 744.700,A 0.000,B 0.000,C 90.000,E1 341.945} C_DIS
LIN {X -0.017,Y -484.231,Z 744.698,A 0.000,B 0.000,C 90.000,E1 341.583} C_DIS
LIN {X -0.057,Y -488.045,Z 744.695,A 0.000,B 0.000,C 90.000,E1 341.094} C_DIS
LIN {X -0.150,Y -492.382,Z 744.693,A 0.000,B 0.000,C 90.000,E1 340.678} C_DIS
LIN {X 0.062,Y -497.885,Z 744.690,A 0.000,B 0.000,C 90.000,E1 340.188} C_DIS
LIN {X 0.128,Y -508.283,Z 744.686,A 0.000,B 0.000,C 90.000,E1 339.444} C_DIS
LIN {X -0.170,Y -524.353,Z 744.680,A 0.000,B 0.000,C 90.000,E1 338.465} C_DIS
LIN {X -0.208,Y -535.554,Z 744.677,A 0.000,B 0.000,C 90.000,E1 337.794} C_DIS
LIN {X -0.090,Y -543.355,Z 744.674,A 0.000,B 0.000,C 90.000,E1 337.283} C_DIS
LIN {X -0.001,Y -550.751,Z 744.671,A 0.000,B 0.000,C 90.000,E1 336.741} C_DIS
LIN {X -0.081,Y -556.244,Z 744.668,A 0.000,B 0.000,C 90.000,E1 336.282} C_DIS
LIN {X -0.161,Y -561.507,Z 744.665,A 0.000,B 0.000,C 90.000,E1 335.793} C_DIS
LIN {X 0.194,Y -567.776,Z 744.662,A 0.000,B 0.000,C 90.000,E1 335.101} C_DIS
LIN {X 0.251,Y -575.083,Z 744.657,A 0.000,B 0.000,C 90.000,E1 334.280} C_DIS
LIN {X -0.131,Y -580.863,Z 744.654,A 0.000,B 0.000,C 90.000,E1 333.640} C_DIS
LIN {X 0.057,Y -587.341,Z 744.649,A 0.000,B 0.000,C 90.000,E1 332.820} C_DIS
LIN {X -0.055,Y -594.640,Z 744.644,A 0.000,B 0.000,C 90.000,E1 331.897} C_DIS
LIN {X -0.146,Y -603.467,Z 744.637,A 0.000,B 0.000,C 90.000,E1 330.717} C_DIS
LIN {X -0.055,Y -609.973,Z 744.632,A 0.000,B 0.000,C 90.000,E1 329.793} C_DIS
LIN {X 0.110,Y -616.113,Z 744.627,A 0.000,B 0.000,C 90.000,E1 328.869} C_DIS
LIN {X -0.190,Y -622.693,Z 744.621,A 0.000,B 0.000,C 90.000,E1 327.867} C_DIS
LIN {X -0.072,Y -628.109,Z 744.616,A 0.000,B 0.000,C 90.000,E1 326.962} C_DIS
LIN {X -0.238,Y -632.415,Z 744.612,A 0.000,B 0.000,C 90.000,E1 326.215} C_DIS
LIN {X 0.014,Y -638.019,Z 744.607,A 0.000,B 0.000,C 90.000,E1 325.182} C_DIS
LIN {X 0.307,Y -641.911,Z 744.602,A 0.000,B 0.000,C 90.000,E1 324.402} C_DIS
LIN {X 0.178,Y -647.404,Z 744.596,A 0.000,B 0.000,C 90.000,E1 323.290} C_DIS
LIN {X -0.035,Y -651.982,Z 744.591,A 0.000,B 0.000,C 90.000,E1 322.316} C_DIS
LIN {X -0.072,Y -656.202,Z 744.585,A 0.000,B 0.000,C 90.000,E1 321.331} C_DIS
LIN {X -0.123,Y -659.206,Z 744.581,A 0.000,B 0.000,C 90.000,E1 320.598} C_DIS
LIN {X -0.175,Y -662.982,Z 744.576,A 0.000,B 0.000,C 90.000,E1 319.622} C_DIS
LIN {X 0.272,Y -665.729,Z 744.572,A 0.000,B 0.000,C 90.000,E1 318.852} C_DIS
LIN {X -0.191,Y -668.266,Z 744.568,A 0.000,B 0.000,C 90.000,E1 318.162} C_DIS
LIN {X 0.323,Y -671.443,Z 744.562,A 0.000,B 0.000,C 90.000,E1 317.148} C_DIS
LIN {X -0.071,Y -674.471,Z 744.557,A 0.000,B 0.000,C 90.000,E1 316.215} C_DIS
LIN {X 0.074,Y -677.954,Z 744.550,A 0.000,B 0.000,C 90.000,E1 315.000} C_DIS
LIN {X 0.189,Y -679.838,Z 744.546,A 0.000,B 0.000,C 90.000,E1 314.271} C_DIS
LIN {X 0.049,Y -683.915,Z 744.537,A 0.000,B 0.000,C 90.000,E1 312.609} C_DIS
LIN {X -0.193,Y -685.982,Z 744.531,A 0.000,B 0.000,C 90.000,E1 311.676} C_DIS
LIN {X 0.168,Y -688.427,Z 744.525,A 0.000,B 0.000,C 90.000,E1 310.458} C_DIS
LIN {X 0.060,Y -690.003,Z 744.520,A 0.000,B 0.000,C 90.000,E1 309.519} C_DIS
LIN {X -0.124,Y -691.375,Z 744.514,A 0.000,B 0.000,C 90.000,E1 308.588} C_DIS
LIN {X -0.005,Y -692.937,Z 744.508,A 0.000,B 0.000,C 90.000,E1 307.397} C_DIS
LIN {X -0.342,Y -694.474,Z 744.500,A 0.000,B 0.000,C 90.000,E1 306.011} C_DIS
LIN {X -0.159,Y -695.537,Z 744.493,A 0.000,B 0.000,C 90.000,E1 304.818} C_DIS
LIN {X -0.073,Y -696.802,Z 744.484,A 0.000,B 0.000,C 90.000,E1 303.166} C_DIS
LIN {X 0.008,Y -697.933,Z 744.476,A 0.000,B 0.000,C 90.000,E1 301.750} C_DIS
LIN {X 0.195,Y -698.656,Z 744.471,A 0.000,B 0.000,C 90.000,E1 300.797} C_DIS
LIN {X -0.231,Y -698.991,Z 744.467,A 0.000,B 0.000,C 90.000,E1 300.129} C_DIS
LIN {X -0.129,Y -699.366,Z 744.461,A 0.000,B 0.000,C 90.000,E1 298.949} C_DIS
LIN {X 0.247,Y -699.823,Z 744.453,A 0.000,B 0.000,C 90.000,E1 297.513} C_DIS
LIN {X 0.191,Y -700.688,Z 744.441,A 0.000,B 0.000,C 90.000,E1 295.412} C_DIS
LIN {X 0.102,Y -700.791,Z 744.439,A 0.000,B 0.000,C 90.000,E1 294.951} C_DIS
LIN {X 0.081,Y -700.803,Z 744.437,A 0.000,B 0.000,C 90.000,E1 294.719} C_DIS
LIN {X -0.284,Y -700.557,Z 744.436,A 0.000,B 0.000,C 90.000,E1 294.515} C_DIS
LIN {X -0.028,Y -699.671,Z 744.434,A 0.000,B 0.000,C 90.000,E1 294.027} C_DIS
LIN {X 0.240,Y -698.640,Z 744.432,A 0.000,B 0.000,C 90.000,E1 293.770} C_DIS
LIN {X -0.153,Y -695.439,Z 744.430,A 0.000,B 0.000,C 90.000,E1 293.334} C_DIS
LIN {X -0.026,Y -694.370,Z 744.429,A 0.000,B 0.000,C 90.000,E1 293.206} C_DIS
LIN {X 0.100,Y -692.747,Z 744.428,A 0.000,B 0.000,C 90.000,E1 293.078} C_DIS
LIN {X 0.199,Y -685.441,Z 744.426,A 0.000,B 0.000,C 90.000,E1 292.717} C_DIS
LIN {X 0.198,Y -683.202,Z 744.426,A 0.000,B 0.000,C 90.000,E1 292.642} C_DIS
LIN {X -0.206,Y -676.638,Z 744.425,A 0.000,B 0.000,C 90.000,E1 292.514} C_DIS
LIN {X 0.012,Y -671.087,Z 744.425,A 0.000,B 0.000,C 90.000,E1 292.408} C_DIS
LIN {X -0.009,Y -664.930,Z 744.424,A 0.000,B 0.000,C 90.000,E1 292.333} C_DIS
LIN {X 0.219,Y -656.544,Z 744.424,A 0.000,B 0.000,C 90.000,E1 292.206} C_DIS
LIN {X -0.184,Y -645.884,Z 744.423,A 0.000,B 0.000,C 90.000,E1 292.078} C_DIS
LIN {X -0.236,Y -636.308,Z 744.422,A 0.000,B 0.000,C 90.000,E1 291.897} C_DIS
LIN {X -0.236,Y -622.649,Z 744.420,A 0.000,B 0.000,C 90.000,E1 291.589} C_DIS
LIN {X -0.091,Y -609.021,Z 744.418,A 0.000,B 0.000,C 90.000,E1 291.227} C_DIS
LIN {X 0.228,Y -577.603,Z 744.413,A 0.000,B 0.000,C 90.000,E1 290.301} C_DIS
LIN {X -0.034,Y -572.050,Z 744.412,A 0.000,B 0.000,C 90.000,E1 290.174} C_DIS
LIN {X 0.355,Y -566.677,Z 744.411,A 0.000,B 0.000,C 90.000,E1 289.993} C_DIS
LIN {X 0.257,Y -561.350,Z 744.410,A 0.000,B 0.000,C 90.000,E1 289.812} C_DIS
LIN {X -0.253,Y -557.031,Z 744.409,A 0.000,B 0.000,C 90.000,E1 289.631} C_DIS
LIN {X 0.217,Y -556.938,Z 744.409,A 0.000,B 0.000,C 90.000,E1 289.577} C_DIS
LIN {X -0.232,Y -555.691,Z 744.408,A 0.000,B 0.000,C 90.000,E1 289.450} C_DIS
LIN {X -0.274,Y -555.677,Z 744.408,A 0.000,B 0.000,C 90.000,E1 289.450} C_DIS
LIN {X -0.074,Y -554.976,Z 744.406,A 0.000,B 0.000,C 90.000,E1 289.033} C_DIS
LIN {X 0.199,Y -554.213,Z 744.394,A 0.000,B 0.000,C 90.000,E1 286.913} C_DIS
LIN {X 0.253,Y -553.454,Z 744.383,A 0.000,B 0.000,C 90.000,E1 284.954} C_DIS
LIN {X 0.157,Y -552.812,Z 744.372,A 0.000,B 0.000,C 90.000,E1 283.008} C_DIS
LIN {X -0.195,Y -552.259,Z 744.363,A 0.000,B 0.000,C 90.000,E1 281.366} C_DIS
LIN {X -0.142,Y -551.792,Z 744.355,A 0.000,B 0.000,C 90.000,E1 279.962} C_DIS
LIN {X -0.201,Y -551.111,Z 744.348,A 0.000,B 0.000,C 90.000,E1 278.568} C_DIS
LIN {X -0.246,Y -550.333,Z 744.338,A 0.000,B 0.000,C 90.000,E1 276.891} C_DIS
LIN {X 0.174,Y -549.564,Z 744.329,A 0.000,B 0.000,C 90.000,E1 275.163} C_DIS
LIN {X 0.109,Y -548.381,Z 744.316,A 0.000,B 0.000,C 90.000,E1 272.922} C_DIS
LIN {X -0.091,Y -547.394,Z 744.305,A 0.000,B 0.000,C 90.000,E1 270.974} C_DIS
LIN {X 0.093,Y -546.710,Z 744.299,A 0.000,B 0.000,C 90.000,E1 269.828} C_DIS
LIN {X -0.144,Y -545.406,Z 744.288,A 0.000,B 0.000,C 90.000,E1 267.879} C_DIS
LIN {X 0.160,Y -544.198,Z 744.277,A 0.000,B 0.000,C 90.000,E1 265.869} C_DIS
LIN {X -0.162,Y -543.227,Z 744.269,A 0.000,B 0.000,C 90.000,E1 264.489} C_DIS
LIN {X 0.019,Y -542.445,Z 744.263,A 0.000,B 0.000,C 90.000,E1 263.337} C_DIS
LIN {X -0.205,Y -541.067,Z 744.254,A 0.000,B 0.000,C 90.000,E1 261.659} C_DIS
LIN {X 0.066,Y -539.661,Z 744.244,A 0.000,B 0.000,C 90.000,E1 259.926} C_DIS
LIN {X -0.046,Y -538.236,Z 744.235,A 0.000,B 0.000,C 90.000,E1 258.229} C_DIS
LIN {X 0.151,Y -537.581,Z 744.230,A 0.000,B 0.000,C 90.000,E1 257.353} C_DIS
LIN {X 0.056,Y -536.289,Z 744.222,A 0.000,B 0.000,C 90.000,E1 255.936} C_DIS
LIN {X -0.062,Y -534.742,Z 744.214,A 0.000,B 0.000,C 90.000,E1 254.519} C_DIS
LIN {X 0.155,Y -532.555,Z 744.203,A 0.000,B 0.000,C 90.000,E1 252.489} C_DIS
LIN {X -0.236,Y -531.025,Z 744.195,A 0.000,B 0.000,C 90.000,E1 251.094} C_DIS
LIN {X 0.027,Y -528.689,Z 744.185,A 0.000,B 0.000,C 90.000,E1 249.337} C_DIS
LIN {X -0.052,Y -526.710,Z 744.177,A 0.000,B 0.000,C 90.000,E1 247.901} C_DIS
LIN {X -0.196,Y -524.065,Z 744.168,A 0.000,B 0.000,C 90.000,E1 246.177} C_DIS
LIN {X 0.182,Y -522.192,Z 744.161,A 0.000,B 0.000,C 90.000,E1 244.973} C_DIS
LIN {X 0.209,Y -519.815,Z 744.153,A 0.000,B 0.000,C 90.000,E1 243.512} C_DIS
LIN {X 0.056,Y -517.727,Z 744.147,A 0.000,B 0.000,C 90.000,E1 242.359} C_DIS
LIN {X -0.227,Y -514.863,Z 744.138,A 0.000,B 0.000,C 90.000,E1 240.923} C_DIS
LIN {X 0.044,Y -511.435,Z 744.129,A 0.000,B 0.000,C 90.000,E1 239.125} C_DIS
LIN {X 0.000,Y -509.128,Z 744.122,A 0.000,B 0.000,C 90.000,E1 237.946} C_DIS
LIN {X 0.031,Y -506.594,Z 744.115,A 0.000,B 0.000,C 90.000,E1 236.755} C_DIS
LIN {X 0.060,Y -503.321,Z 744.107,A 0.000,B 0.000,C 90.000,E1 235.261} C_DIS
LIN {X 0.013,Y -500.532,Z 744.100,A 0.000,B 0.000,C 90.000,E1 234.069} C_DIS
LIN {X 0.219,Y -497.507,Z 744.094,A 0.000,B 0.000,C 90.000,E1 232.844} C_DIS
LIN {X 0.094,Y -492.956,Z 744.084,A 0.000,B 0.000,C 90.000,E1 231.045} C_DIS
LIN {X -0.057,Y -487.909,Z 744.072,A 0.000,B 0.000,C 90.000,E1 228.933} C_DIS
LIN {X 0.178,Y -483.797,Z 744.062,A 0.000,B 0.000,C 90.000,E1 227.067} C_DIS
LIN {X -0.031,Y -479.843,Z 744.051,A 0.000,B 0.000,C 90.000,E1 225.243} C_DIS
LIN {X 0.003,Y -475.936,Z 744.041,A 0.000,B 0.000,C 90.000,E1 223.380} C_DIS
LIN {X -0.040,Y -471.866,Z 744.031,A 0.000,B 0.000,C 90.000,E1 221.515} C_DIS
LIN {X -0.131,Y -467.669,Z 744.020,A 0.000,B 0.000,C 90.000,E1 219.644} C_DIS
LIN {X -0.201,Y -462.892,Z 744.008,A 0.000,B 0.000,C 90.000,E1 217.443} C_DIS
LIN {X -0.202,Y -457.615,Z 743.994,A 0.000,B 0.000,C 90.000,E1 214.898} C_DIS
LIN {X -0.166,Y -454.429,Z 743.985,A 0.000,B 0.000,C 90.000,E1 213.293} C_DIS
LIN {X 0.029,Y -450.833,Z 743.974,A 0.000,B 0.000,C 90.000,E1 211.337} C_DIS
LIN {X -0.020,Y -446.651,Z 743.962,A 0.000,B 0.000,C 90.000,E1 209.077} C_DIS
LIN {X -0.020,Y -442.402,Z 743.949,A 0.000,B 0.000,C 90.000,E1 206.796} C_DIS
LIN {X 0.149,Y -439.952,Z 743.942,A 0.000,B 0.000,C 90.000,E1 205.463} C_DIS
LIN {X 0.115,Y -436.870,Z 743.932,A 0.000,B 0.000,C 90.000,E1 203.823} C_DIS
LIN {X 0.074,Y -433.174,Z 743.921,A 0.000,B 0.000,C 90.000,E1 201.844} C_DIS
LIN {X -0.184,Y -428.146,Z 743.907,A 0.000,B 0.000,C 90.000,E1 199.214} C_DIS
LIN {X -0.175,Y -425.706,Z 743.899,A 0.000,B 0.000,C 90.000,E1 197.873} C_DIS
LIN {X 0.080,Y -421.082,Z 743.886,A 0.000,B 0.000,C 90.000,E1 195.481} C_DIS
LIN {X -0.016,Y -416.679,Z 743.873,A 0.000,B 0.000,C 90.000,E1 193.119} C_DIS
LIN {X -0.131,Y -414.285,Z 743.865,A 0.000,B 0.000,C 90.000,E1 191.771} C_DIS
LIN {X 0.153,Y -411.260,Z 743.856,A 0.000,B 0.000,C 90.000,E1 190.018} C_DIS
LIN {X -0.130,Y -408.960,Z 743.848,A 0.000,B 0.000,C 90.000,E1 188.681} C_DIS
LIN {X -0.120,Y -405.040,Z 743.835,A 0.000,B 0.000,C 90.000,E1 186.258} C_DIS
LIN {X -0.154,Y -403.417,Z 743.829,A 0.000,B 0.000,C 90.000,E1 185.220} C_DIS
LIN {X 0.078,Y -400.424,Z 743.817,A 0.000,B 0.000,C 90.000,E1 183.094} C_DIS
LIN {X -0.100,Y -398.538,Z 743.810,A 0.000,B 0.000,C 90.000,E1 181.718} C_DIS
LIN {X 0.118,Y -394.447,Z 743.790,A 0.000,B 0.000,C 90.000,E1 178.165} C_DIS
LIN {X -0.100,Y -391.271,Z 743.772,A 0.000,B 0.000,C 90.000,E1 175.008} C_DIS
LIN {X 0.081,Y -387.946,Z 743.743,A 0.000,B 0.000,C 90.000,E1 169.634} C_DIS
LIN {X -0.146,Y -387.010,Z 743.731,A 0.000,B 0.000,C 90.000,E1 167.521} C_DIS
LIN {X 0.078,Y -386.170,Z 743.719,A 0.000,B 0.000,C 90.000,E1 165.338} C_DIS
LIN {X 0.029,Y -385.507,Z 743.705,A 0.000,B 0.000,C 90.000,E1 162.834} C_DIS
LIN {X 0.060,Y -384.982,Z 743.691,A 0.000,B 0.000,C 90.000,E1 160.315} C_DIS
LIN {X -0.079,Y -384.705,Z 743.681,A 0.000,B 0.000,C 90.000,E1 158.539} C_DIS
LIN {X -0.099,Y -384.380,Z 743.665,A 0.000,B 0.000,C 90.000,E1 155.665} C_DIS
LIN {X 0.006,Y -385.949,Z 743.631,A 0.000,B 0.000,C 90.000,E1 149.537} C_DIS
LIN {X 0.079,Y -387.310,Z 743.619,A 0.000,B 0.000,C 90.000,E1 147.375} C_DIS
LIN {X -0.113,Y -392.373,Z 743.593,A 0.000,B 0.000,C 90.000,E1 142.763} C_DIS
LIN {X -0.022,Y -394.853,Z 743.585,A 0.000,B 0.000,C 90.000,E1 141.331} C_DIS
LIN {X -0.147,Y -396.408,Z 743.581,A 0.000,B 0.000,C 90.000,E1 140.642} C_DIS
LIN {X -0.051,Y -397.298,Z 743.579,A 0.000,B 0.000,C 90.000,E1 140.275} C_DIS
LIN {X 0.052,Y -400.153,Z 743.574,A 0.000,B 0.000,C 90.000,E1 139.380} C_DIS
LIN {X 0.068,Y -402.473,Z 743.572,A 0.000,B 0.000,C 90.000,E1 138.852} C_DIS
LIN {X 0.013,Y -406.619,Z 743.568,A 0.000,B 0.000,C 90.000,E1 138.162} C_DIS
LIN {X -0.058,Y -409.691,Z 743.565,A 0.000,B 0.000,C 90.000,E1 137.757} C_DIS
LIN {X 0.101,Y -417.676,Z 743.560,A 0.000,B 0.000,C 90.000,E1 136.863} C_DIS
LIN {X -0.024,Y -434.961,Z 743.551,A 0.000,B 0.000,C 90.000,E1 135.121} C_DIS
LIN {X 0.189,Y -445.082,Z 743.545,A 0.000,B 0.000,C 90.000,E1 134.109} C_DIS
LIN {X 0.107,Y -453.881,Z 743.540,A 0.000,B 0.000,C 90.000,E1 133.257} C_DIS
LIN {X 0.127,Y -459.490,Z 743.537,A 0.000,B 0.000,C 90.000,E1 132.690} C_DIS
LIN {X 0.045,Y -465.105,Z 743.534,A 0.000,B 0.000,C 90.000,E1 132.123} C_DIS
LIN {X -0.032,Y -473.322,Z 743.529,A 0.000,B 0.000,C 90.000,E1 131.272} C_DIS
LIN {X 0.142,Y -479.824,Z 743.525,A 0.000,B 0.000,C 90.000,E1 130.539} C_DIS
LIN {X -0.143,Y -487.442,Z 743.521,A 0.000,B 0.000,C 90.000,E1 129.725} C_DIS
LIN {X -0.143,Y -493.583,Z 743.517,A 0.000,B 0.000,C 90.000,E1 128.991} C_DIS
LIN {X -0.031,Y -495.882,Z 743.515,A 0.000,B 0.000,C 90.000,E1 128.705} C_DIS
LIN {X 0.118,Y -501.603,Z 743.511,A 0.000,B 0.000,C 90.000,E1 127.935} C_DIS
LIN {X -0.217,Y -504.939,Z 743.508,A 0.000,B 0.000,C 90.000,E1 127.523} C_DIS
LIN {X 0.280,Y -509.050,Z 743.505,A 0.000,B 0.000,C 90.000,E1 126.870} C_DIS
LIN {X 0.017,Y -514.720,Z 743.500,A 0.000,B 0.000,C 90.000,E1 126.011} C_DIS
LIN {X -0.244,Y -517.441,Z 743.498,A 0.000,B 0.000,C 90.000,E1 125.598} C_DIS
LIN {X 0.231,Y -520.051,Z 743.495,A 0.000,B 0.000,C 90.000,E1 125.105} C_DIS
LIN {X 0.076,Y -524.609,Z 743.490,A 0.000,B 0.000,C 90.000,E1 124.246} C_DIS
LIN {X 0.270,Y -528.139,Z 743.486,A 0.000,B 0.000,C 90.000,E1 123.499} C_DIS
LIN {X 0.328,Y -533.356,Z 743.480,A 0.000,B 0.000,C 90.000,E1 122.339} C_DIS
LIN {X -0.138,Y -537.618,Z 743.474,A 0.000,B 0.000,C 90.000,E1 121.386} C_DIS
LIN {X -0.242,Y -541.067,Z 743.470,A 0.000,B 0.000,C 90.000,E1 120.541} C_DIS
LIN {X -0.031,Y -544.352,Z 743.465,A 0.000,B 0.000,C 90.000,E1 119.667} C_DIS
LIN {X -0.054,Y -547.466,Z 743.460,A 0.000,B 0.000,C 90.000,E1 118.821} C_DIS
LIN {X -0.278,Y -551.317,Z 743.454,A 0.000,B 0.000,C 90.000,E1 117.719} C_DIS
LIN {X 0.045,Y -554.856,Z 743.448,A 0.000,B 0.000,C 90.000,E1 116.565} C_DIS
LIN {X -0.082,Y -557.761,Z 743.441,A 0.000,B 0.000,C 90.000,E1 115.463} C_DIS
LIN {X -0.211,Y -559.586,Z 743.437,A 0.000,B 0.000,C 90.000,E1 114.643} C_DIS
LIN {X -0.115,Y -560.713,Z 743.434,A 0.000,B 0.000,C 90.000,E1 114.079} C_DIS
LIN {X 0.101,Y -562.539,Z 743.428,A 0.000,B 0.000,C 90.000,E1 112.950} C_DIS
LIN {X -0.074,Y -564.509,Z 743.420,A 0.000,B 0.000,C 90.000,E1 111.589} C_DIS
LIN {X -0.085,Y -566.833,Z 743.411,A 0.000,B 0.000,C 90.000,E1 109.939} C_DIS
LIN {X 0.149,Y -568.615,Z 743.403,A 0.000,B 0.000,C 90.000,E1 108.544} C_DIS
LIN {X 0.068,Y -569.912,Z 743.397,A 0.000,B 0.000,C 90.000,E1 107.457} C_DIS
LIN {X 0.178,Y -571.531,Z 743.389,A 0.000,B 0.000,C 90.000,E1 106.079} C_DIS
LIN {X -0.202,Y -573.312,Z 743.380,A 0.000,B 0.000,C 90.000,E1 104.481} C_DIS
LIN {X -0.188,Y -574.870,Z 743.373,A 0.000,B 0.000,C 90.000,E1 103.119} C_DIS
LIN {X 0.140,Y -577.024,Z 743.362,A 0.000,B 0.000,C 90.000,E1 101.186} C_DIS
LIN {X 0.193,Y -578.776,Z 743.353,A 0.000,B 0.000,C 90.000,E1 99.557} C_DIS
LIN {X 0.054,Y -580.093,Z 743.346,A 0.000,B 0.000,C 90.000,E1 98.219} C_DIS
LIN {X -0.150,Y -581.408,Z 743.338,A 0.000,B 0.000,C 90.000,E1 96.891} C_DIS
LIN {X -0.176,Y -582.836,Z 743.329,A 0.000,B 0.000,C 90.000,E1 95.277} C_DIS
LIN {X 0.184,Y -583.917,Z 743.322,A 0.000,B 0.000,C 90.000,E1 93.898} C_DIS
LIN {X -0.057,Y -584.941,Z 743.314,A 0.000,B 0.000,C 90.000,E1 92.579} C_DIS
LIN {X -0.280,Y -585.852,Z 743.307,A 0.000,B 0.000,C 90.000,E1 91.260} C_DIS
LIN {X 0.278,Y -586.710,Z 743.298,A 0.000,B 0.000,C 90.000,E1 89.599} C_DIS
LIN {X 0.281,Y -587.335,Z 743.289,A 0.000,B 0.000,C 90.000,E1 87.993} C_DIS
LIN {X -0.291,Y -587.873,Z 743.280,A 0.000,B 0.000,C 90.000,E1 86.445} C_DIS
LIN {X 0.164,Y -588.142,Z 743.273,A 0.000,B 0.000,C 90.000,E1 85.065} C_DIS
LIN {X 0.214,Y -588.312,Z 743.264,A 0.000,B 0.000,C 90.000,E1 83.457} C_DIS
LIN {X 0.144,Y -588.342,Z 743.256,A 0.000,B 0.000,C 90.000,E1 82.129} C_DIS
LIN {X -0.093,Y -588.310,Z 743.250,A 0.000,B 0.000,C 90.000,E1 81.084} C_DIS
LIN {X 0.254,Y -588.158,Z 743.245,A 0.000,B 0.000,C 90.000,E1 79.982} C_DIS
LIN {X -0.055,Y -587.641,Z 743.236,A 0.000,B 0.000,C 90.000,E1 78.409} C_DIS
LIN {X 0.063,Y -587.118,Z 743.228,A 0.000,B 0.000,C 90.000,E1 77.061} C_DIS
LIN {X 0.060,Y -586.625,Z 743.222,A 0.000,B 0.000,C 90.000,E1 75.992} C_DIS
LIN {X -0.018,Y -585.773,Z 743.213,A 0.000,B 0.000,C 90.000,E1 74.393} C_DIS
LIN {X 0.040,Y -584.714,Z 743.204,A 0.000,B 0.000,C 90.000,E1 72.779} C_DIS
LIN {X -0.150,Y -583.674,Z 743.197,A 0.000,B 0.000,C 90.000,E1 71.456} C_DIS
LIN {X -0.170,Y -582.575,Z 743.190,A 0.000,B 0.000,C 90.000,E1 70.115} C_DIS
LIN {X -0.064,Y -581.580,Z 743.184,A 0.000,B 0.000,C 90.000,E1 69.028} C_DIS
LIN {X 0.227,Y -580.486,Z 743.177,A 0.000,B 0.000,C 90.000,E1 67.922} C_DIS
LIN {X -0.037,Y -579.253,Z 743.172,A 0.000,B 0.000,C 90.000,E1 66.869} C_DIS
LIN {X -0.086,Y -577.856,Z 743.166,A 0.000,B 0.000,C 90.000,E1 65.793} C_DIS
LIN {X -0.147,Y -576.320,Z 743.159,A 0.000,B 0.000,C 90.000,E1 64.717} C_DIS
LIN {X -0.231,Y -574.526,Z 743.154,A 0.000,B 0.000,C 90.000,E1 63.640} C_DIS
LIN {X -0.083,Y -572.558,Z 743.147,A 0.000,B 0.000,C 90.000,E1 62.538} C_DIS
LIN {X -0.066,Y -570.848,Z 743.143,A 0.000,B 0.000,C 90.000,E1 61.719} C_DIS
LIN {X -0.302,Y -568.945,Z 743.138,A 0.000,B 0.000,C 90.000,E1 60.923} C_DIS
LIN {X 0.040,Y -566.092,Z 743.132,A 0.000,B 0.000,C 90.000,E1 59.793} C_DIS
LIN {X -0.237,Y -563.749,Z 743.128,A 0.000,B 0.000,C 90.000,E1 58.997} C_DIS
LIN {X 0.234,Y -561.242,Z 743.123,A 0.000,B 0.000,C 90.000,E1 58.122} C_DIS
LIN {X -0.100,Y -558.458,Z 743.118,A 0.000,B 0.000,C 90.000,E1 57.327} C_DIS
LIN {X -0.162,Y -555.404,Z 743.114,A 0.000,B 0.000,C 90.000,E1 56.501} C_DIS
LIN {X -0.255,Y -551.965,Z 743.109,A 0.000,B 0.000,C 90.000,E1 55.674} C_DIS
LIN {X -0.127,Y -549.523,Z 743.106,A 0.000,B 0.000,C 90.000,E1 55.102} C_DIS
LIN {X -0.268,Y -545.366,Z 743.101,A 0.000,B 0.000,C 90.000,E1 54.276} C_DIS
LIN {X -0.014,Y -541.635,Z 743.097,A 0.000,B 0.000,C 90.000,E1 53.543} C_DIS
LIN {X -0.133,Y -539.314,Z 743.095,A 0.000,B 0.000,C 90.000,E1 53.130} C_DIS
LIN {X 0.067,Y -534.878,Z 743.091,A 0.000,B 0.000,C 90.000,E1 52.396} C_DIS
LIN {X 0.106,Y -531.029,Z 743.088,A 0.000,B 0.000,C 90.000,E1 51.823} C_DIS
LIN {X 0.187,Y -526.849,Z 743.085,A 0.000,B 0.000,C 90.000,E1 51.251} C_DIS
LIN {X -0.207,Y -522.073,Z 743.082,A 0.000,B 0.000,C 90.000,E1 50.723} C_DIS
LIN {X -0.054,Y -518.161,Z 743.079,A 0.000,B 0.000,C 90.000,E1 50.275} C_DIS
LIN {X 0.095,Y -512.480,Z 743.076,A 0.000,B 0.000,C 90.000,E1 49.703} C_DIS
LIN {X 0.168,Y -508.121,Z 743.074,A 0.000,B 0.000,C 90.000,E1 49.299} C_DIS
LIN {X -0.280,Y -501.991,Z 743.071,A 0.000,B 0.000,C 90.000,E1 48.852} C_DIS
LIN {X -0.063,Y -494.105,Z 743.068,A 0.000,B 0.000,C 90.000,E1 48.243} C_DIS
LIN {X 0.047,Y -486.081,Z 743.065,A 0.000,B 0.000,C 90.000,E1 47.676} C_DIS
LIN {X -0.128,Y -472.997,Z 743.060,A 0.000,B 0.000,C 90.000,E1 46.863} C_DIS
LIN {X -0.182,Y -455.002,Z 743.054,A 0.000,B 0.000,C 90.000,E1 45.729} C_DIS
LIN {X 0.094,Y -432.405,Z 743.046,A 0.000,B 0.000,C 90.000,E1 44.190} C_DIS
LIN {X -0.087,Y -419.856,Z 743.041,A 0.000,B 0.000,C 90.000,E1 43.299} C_DIS
LIN {X -0.023,Y -414.184,Z 743.038,A 0.000,B 0.000,C 90.000,E1 42.813} C_DIS
LIN {X 0.092,Y -413.898,Z 743.038,A 0.000,B 0.000,C 90.000,E1 42.771} C_DIS
LIN {X 0.061,Y -413.883,Z 743.038,A 0.000,B 0.000,C 90.000,E1 42.771} C_DIS
LIN {X 0.104,Y -405.672,Z 743.013,A 0.000,B 0.000,C 90.000,E1 38.382} C_DIS
LIN {X 0.082,Y -402.644,Z 743.006,A 0.000,B 0.000,C 90.000,E1 36.996} C_DIS
LIN {X -0.032,Y -402.583,Z 743.004,A 0.000,B 0.000,C 90.000,E1 36.664} C_DIS
LIN {X 0.141,Y -403.106,Z 742.986,A 0.000,B 0.000,C 90.000,E1 33.499} C_DIS
LIN {X -0.004,Y -404.405,Z 742.969,A 0.000,B 0.000,C 90.000,E1 30.384} C_DIS
LIN {X -0.011,Y -406.000,Z 742.951,A 0.000,B 0.000,C 90.000,E1 27.257} C_DIS
LIN {X 0.033,Y -408.027,Z 742.934,A 0.000,B 0.000,C 90.000,E1 24.131} C_DIS
LIN {X 0.128,Y -410.386,Z 742.919,A 0.000,B 0.000,C 90.000,E1 21.354} C_DIS
LIN {X -0.082,Y -414.137,Z 742.900,A 0.000,B 0.000,C 90.000,E1 17.946} C_DIS
LIN {X 0.227,Y -418.193,Z 742.883,A 0.000,B 0.000,C 90.000,E1 14.828} C_DIS
LIN {X -0.111,Y -420.713,Z 742.873,A 0.000,B 0.000,C 90.000,E1 13.175} C_DIS
LIN {X -0.004,Y -423.855,Z 742.862,A 0.000,B 0.000,C 90.000,E1 11.130} C_DIS
LIN {X 0.110,Y -427.027,Z 742.851,A 0.000,B 0.000,C 90.000,E1 9.095} C_DIS
LIN {X -0.190,Y -430.183,Z 742.839,A 0.000,B 0.000,C 90.000,E1 7.125} C_DIS
LIN {X 0.145,Y -434.535,Z 742.825,A 0.000,B 0.000,C 90.000,E1 4.416} C_DIS
LIN {X -0.013,Y -438.592,Z 742.812,A 0.000,B 0.000,C 90.000,E1 2.121} C_DIS
LIN {X 0.122,Y -441.715,Z 742.803,A 0.000,B 0.000,C 90.000,E1 0.458} C_DIS
LIN {X 0.088,Y -446.865,Z 742.788,A 0.000,B 0.000,C 90.000,E1 357.822} C_DIS
LIN {X 0.122,Y -450.974,Z 742.777,A 0.000,B 0.000,C 90.000,E1 355.869} C_DIS
LIN {X -0.001,Y -455.996,Z 742.765,A 0.000,B 0.000,C 90.000,E1 353.628} C_DIS
LIN {X 0.150,Y -459.580,Z 742.756,A 0.000,B 0.000,C 90.000,E1 352.008} C_DIS
LIN {X 0.128,Y -462.339,Z 742.749,A 0.000,B 0.000,C 90.000,E1 350.735} C_DIS
LIN {X 0.022,Y -465.518,Z 742.740,A 0.000,B 0.000,C 90.000,E1 349.162} C_DIS
LIN {X 0.163,Y -467.870,Z 742.733,A 0.000,B 0.000,C 90.000,E1 347.881} C_DIS
LIN {X -0.208,Y -470.784,Z 742.724,A 0.000,B 0.000,C 90.000,E1 346.353} C_DIS
LIN {X 0.242,Y -475.532,Z 742.710,A 0.000,B 0.000,C 90.000,E1 343.795} C_DIS
LIN {X 0.037,Y -477.056,Z 742.707,A 0.000,B 0.000,C 90.000,E1 343.196} C_DIS
LIN {X -0.159,Y -478.905,Z 742.703,A 0.000,B 0.000,C 90.000,E1 342.598} C_DIS
LIN {X -0.107,Y -480.678,Z 742.701,A 0.000,B 0.000,C 90.000,E1 342.127} C_DIS
LIN {X -0.121,Y -482.118,Z 742.699,A 0.000,B 0.000,C 90.000,E1 341.819} C_DIS
LIN {X 0.031,Y -484.374,Z 742.697,A 0.000,B 0.000,C 90.000,E1 341.402} C_DIS
LIN {X 0.031,Y -486.587,Z 742.695,A 0.000,B 0.000,C 90.000,E1 341.094} C_DIS
LIN {X 0.043,Y -489.135,Z 742.693,A 0.000,B 0.000,C 90.000,E1 340.786} C_DIS
LIN {X -0.046,Y -496.453,Z 742.690,A 0.000,B 0.000,C 90.000,E1 340.115} C_DIS
LIN {X 0.204,Y -505.128,Z 742.686,A 0.000,B 0.000,C 90.000,E1 339.444} C_DIS
LIN {X 0.101,Y -522.618,Z 742.680,A 0.000,B 0.000,C 90.000,E1 338.337} C_DIS
LIN {X 0.051,Y -533.908,Z 742.676,A 0.000,B 0.000,C 90.000,E1 337.667} C_DIS
LIN {X 0.008,Y -540.225,Z 742.674,A 0.000,B 0.000,C 90.000,E1 337.283} C_DIS
LIN {X 0.169,Y -547.820,Z 742.671,A 0.000,B 0.000,C 90.000,E1 336.741} C_DIS
LIN {X -0.056,Y -551.998,Z 742.669,A 0.000,B 0.000,C 90.000,E1 336.433} C_DIS
LIN {X 0.139,Y -556.129,Z 742.667,A 0.000,B 0.000,C 90.000,E1 336.049} C_DIS
LIN {X 0.240,Y -561.510,Z 742.664,A 0.000,B 0.000,C 90.000,E1 335.537} C_DIS
LIN {X -0.161,Y -567.849,Z 742.661,A 0.000,B 0.000,C 90.000,E1 334.921} C_DIS
LIN {X 0.139,Y -575.160,Z 742.656,A 0.000,B 0.000,C 90.000,E1 334.076} C_DIS
LIN {X 0.280,Y -580.980,Z 742.652,A 0.000,B 0.000,C 90.000,E1 333.384} C_DIS
LIN {X -0.053,Y -586.500,Z 742.649,A 0.000,B 0.000,C 90.000,E1 332.743} C_DIS
LIN {X 0.352,Y -593.842,Z 742.643,A 0.000,B 0.000,C 90.000,E1 331.769} C_DIS
LIN {X 0.254,Y -602.735,Z 742.637,A 0.000,B 0.000,C 90.000,E1 330.589} C_DIS
LIN {X 0.059,Y -608.407,Z 742.632,A 0.000,B 0.000,C 90.000,E1 329.822} C_DIS
LIN {X -0.008,Y -614.659,Z 742.627,A 0.000,B 0.000,C 90.000,E1 328.918} C_DIS
LIN {X 0.202,Y -621.361,Z 742.622,A 0.000,B 0.000,C 90.000,E1 327.867} C_DIS
LIN {X 0.306,Y -627.627,Z 742.616,A 0.000,B 0.000,C 90.000,E1 326.834} C_DIS
LIN {X -0.380,Y -633.473,Z 742.610,A 0.000,B 0.000,C 90.000,E1 325.881} C_DIS
LIN {X -0.121,Y -638.992,Z 742.605,A 0.000,B 0.000,C 90.000,E1 324.848} C_DIS
LIN {X 0.177,Y -642.786,Z 742.601,A 0.000,B 0.000,C 90.000,E1 324.069} C_DIS
LIN {X 0.016,Y -647.123,Z 742.596,A 0.000,B 0.000,C 90.000,E1 323.210} C_DIS
LIN {X 0.318,Y -651.755,Z 742.590,A 0.000,B 0.000,C 90.000,E1 322.190} C_DIS
LIN {X 0.220,Y -657.050,Z 742.583,A 0.000,B 0.000,C 90.000,E1 320.964} C_DIS
LIN {X -0.330,Y -660.066,Z 742.579,A 0.000,B 0.000,C 90.000,E1 320.275} C_DIS
LIN {X 0.116,Y -664.818,Z 742.572,A 0.000,B 0.000,C 90.000,E1 319.013} C_DIS
LIN {X -0.361,Y -668.208,Z 742.567,A 0.000,B 0.000,C 90.000,E1 318.081} C_DIS
LIN {X 0.152,Y -671.420,Z 742.562,A 0.000,B 0.000,C 90.000,E1 317.067} C_DIS
LIN {X -0.242,Y -674.478,Z 742.556,A 0.000,B 0.000,C 90.000,E1 316.134} C_DIS
LIN {X -0.132,Y -677.307,Z 742.551,A 0.000,B 0.000,C 90.000,E1 315.162} C_DIS
LIN {X -0.023,Y -679.289,Z 742.547,A 0.000,B 0.000,C 90.000,E1 314.433} C_DIS
LIN {X -0.174,Y -683.437,Z 742.538,A 0.000,B 0.000,C 90.000,E1 312.771} C_DIS
LIN {X -0.420,Y -685.613,Z 742.532,A 0.000,B 0.000,C 90.000,E1 311.838} C_DIS
LIN {X -0.065,Y -688.125,Z 742.526,A 0.000,B 0.000,C 90.000,E1 310.620} C_DIS
LIN {X 0.265,Y -689.789,Z 742.520,A 0.000,B 0.000,C 90.000,E1 309.644} C_DIS
LIN {X -0.358,Y -691.241,Z 742.515,A 0.000,B 0.000,C 90.000,E1 308.749} C_DIS
LIN {X 0.184,Y -692.839,Z 742.509,A 0.000,B 0.000,C 90.000,E1 307.523} C_DIS
LIN {X -0.159,Y -694.444,Z 742.501,A 0.000,B 0.000,C 90.000,E1 306.137} C_DIS
LIN {X -0.032,Y -695.326,Z 742.495,A 0.000,B 0.000,C 90.000,E1 305.185} C_DIS
LIN {X -0.177,Y -696.473,Z 742.488,A 0.000,B 0.000,C 90.000,E1 303.785} C_DIS
LIN {X -0.072,Y -697.779,Z 742.479,A 0.000,B 0.000,C 90.000,E1 302.133} C_DIS
LIN {X 0.363,Y -698.720,Z 742.472,A 0.000,B 0.000,C 90.000,E1 300.924} C_DIS
LIN {X -0.065,Y -699.089,Z 742.468,A 0.000,B 0.000,C 90.000,E1 300.256} C_DIS
LIN {X 0.037,Y -699.470,Z 742.462,A 0.000,B 0.000,C 90.000,E1 299.077} C_DIS
LIN {X 0.415,Y -699.900,Z 742.454,A 0.000,B 0.000,C 90.000,E1 297.641} C_DIS
LIN {X 0.087,Y -700.634,Z 742.443,A 0.000,B 0.000,C 90.000,E1 295.796} C_DIS
LIN {X 0.273,Y -700.930,Z 742.440,A 0.000,B 0.000,C 90.000,E1 295.079} C_DIS
LIN {X -0.112,Y -700.900,Z 742.437,A 0.000,B 0.000,C 90.000,E1 294.643} C_DIS
LIN {X 0.144,Y -700.051,Z 742.434,A 0.000,B 0.000,C 90.000,E1 294.155} C_DIS
LIN {X -0.225,Y -699.488,Z 742.433,A 0.000,B 0.000,C 90.000,E1 293.951} C_DIS
LIN {X -0.091,Y -698.910,Z 742.432,A 0.000,B 0.000,C 90.000,E1 293.823} C_DIS
LIN {X 0.026,Y -696.495,Z 742.430,A 0.000,B 0.000,C 90.000,E1 293.462} C_DIS
LIN {X 0.282,Y -694.481,Z 742.429,A 0.000,B 0.000,C 90.000,E1 293.206} C_DIS
LIN {X -0.231,Y -692.987,Z 742.428,A 0.000,B 0.000,C 90.000,E1 293.131} C_DIS
LIN {X 0.141,Y -687.323,Z 742.427,A 0.000,B 0.000,C 90.000,E1 292.823} C_DIS
LIN {X -0.142,Y -685.538,Z 742.426,A 0.000,B 0.000,C 90.000,E1 292.770} C_DIS
LIN {X -0.158,Y -683.355,Z 742.426,A 0.000,B 0.000,C 90.000,E1 292.695} C_DIS
LIN {X 0.055,Y -676.789,Z 742.425,A 0.000,B 0.000,C 90.000,E1 292.514} C_DIS
LIN {X -0.220,Y -672.071,Z 742.425,A 0.000,B 0.000,C 90.000,E1 292.461} C_DIS
LIN {X -0.035,Y -667.903,Z 742.424,A 0.000,B 0.000,C 90.000,E1 292.386} C_DIS
LIN {X -0.197,Y -661.491,Z 742.424,A 0.000,B 0.000,C 90.000,E1 292.333} C_DIS
LIN {X -0.368,Y -648.240,Z 742.423,A 0.000,B 0.000,C 90.000,E1 292.153} C_DIS
LIN {X -0.103,Y -638.521,Z 742.422,A 0.000,B 0.000,C 90.000,E1 291.950} C_DIS
LIN {X -0.190,Y -625.034,Z 742.420,A 0.000,B 0.000,C 90.000,E1 291.663} C_DIS
LIN {X -0.170,Y -608.115,Z 742.418,A 0.000,B 0.000,C 90.000,E1 291.227} C_DIS
LIN {X 0.149,Y -574.879,Z 742.413,A 0.000,B 0.000,C 90.000,E1 290.248} C_DIS
LIN {X 0.055,Y -567.439,Z 742.412,A 0.000,B 0.000,C 90.000,E1 290.066} C_DIS
LIN {X 0.179,Y -560.767,Z 742.410,A 0.000,B 0.000,C 90.000,E1 289.812} C_DIS
LIN {X -0.072,Y -557.001,Z 742.409,A 0.000,B 0.000,C 90.000,E1 289.631} C_DIS
LIN {X -0.126,Y -556.908,Z 742.409,A 0.000,B 0.000,C 90.000,E1 289.631} C_DIS
LIN {X -0.262,Y -555.639,Z 742.408,A 0.000,B 0.000,C 90.000,E1 289.450} C_DIS
LIN {X -0.104,Y -554.945,Z 742.406,A 0.000,B 0.000,C 90.000,E1 289.033} C_DIS
LIN {X 0.068,Y -554.266,Z 742.395,A 0.000,B 0.000,C 90.000,E1 287.149} C_DIS
LIN {X -0.264,Y -553.711,Z 742.388,A 0.000,B 0.000,C 90.000,E1 285.788} C_DIS
LIN {X 0.200,Y -553.117,Z 742.378,A 0.000,B 0.000,C 90.000,E1 284.064} C_DIS
LIN {X 0.270,Y -552.758,Z 742.372,A 0.000,B 0.000,C 90.000,E1 282.939} C_DIS
LIN {X -0.213,Y -552.328,Z 742.364,A 0.000,B 0.000,C 90.000,E1 281.591} C_DIS
LIN {X -0.266,Y -551.860,Z 742.357,A 0.000,B 0.000,C 90.000,E1 280.197} C_DIS
LIN {X 0.226,Y -551.206,Z 742.349,A 0.000,B 0.000,C 90.000,E1 278.746} C_DIS
LIN {X -0.250,Y -550.270,Z 742.338,A 0.000,B 0.000,C 90.000,E1 276.834} C_DIS
LIN {X 0.170,Y -549.508,Z 742.328,A 0.000,B 0.000,C 90.000,E1 275.106} C_DIS
LIN {X -0.019,Y -548.651,Z 742.319,A 0.000,B 0.000,C 90.000,E1 273.440} C_DIS
LIN {X -0.141,Y -547.539,Z 742.307,A 0.000,B 0.000,C 90.000,E1 271.203} C_DIS
LIN {X 0.045,Y -546.870,Z 742.300,A 0.000,B 0.000,C 90.000,E1 270.057} C_DIS
LIN {X 0.262,Y -545.949,Z 742.293,A 0.000,B 0.000,C 90.000,E1 268.625} C_DIS
LIN {X -0.037,Y -544.873,Z 742.283,A 0.000,B 0.000,C 90.000,E1 266.963} C_DIS
LIN {X 0.185,Y -544.013,Z 742.275,A 0.000,B 0.000,C 90.000,E1 265.527} C_DIS
LIN {X -0.148,Y -543.008,Z 742.267,A 0.000,B 0.000,C 90.000,E1 264.147} C_DIS
LIN {X 0.022,Y -542.160,Z 742.261,A 0.000,B 0.000,C 90.000,E1 262.996} C_DIS
LIN {X -0.214,Y -541.057,Z 742.253,A 0.000,B 0.000,C 90.000,E1 261.602} C_DIS
LIN {X 0.148,Y -539.631,Z 742.244,A 0.000,B 0.000,C 90.000,E1 259.859} C_DIS
LIN {X -0.062,Y -538.212,Z 742.234,A 0.000,B 0.000,C 90.000,E1 258.173} C_DIS
LIN {X 0.134,Y -537.555,Z 742.230,A 0.000,B 0.000,C 90.000,E1 257.297} C_DIS
LIN {X 0.036,Y -536.257,Z 742.222,A 0.000,B 0.000,C 90.000,E1 255.880} C_DIS
LIN {X 0.057,Y -534.713,Z 742.214,A 0.000,B 0.000,C 90.000,E1 254.448} C_DIS
LIN {X 0.058,Y -533.132,Z 742.206,A 0.000,B 0.000,C 90.000,E1 253.015} C_DIS
LIN {X 0.023,Y -531.633,Z 742.198,A 0.000,B 0.000,C 90.000,E1 251.583} C_DIS
LIN {X -0.271,Y -530.989,Z 742.195,A 0.000,B 0.000,C 90.000,E1 251.040} C_DIS
LIN {X 0.173,Y -528.633,Z 742.185,A 0.000,B 0.000,C 90.000,E1 249.263} C_DIS
LIN {X -0.098,Y -526.672,Z 742.177,A 0.000,B 0.000,C 90.000,E1 247.847} C_DIS
LIN {X -0.036,Y -524.044,Z 742.167,A 0.000,B 0.000,C 90.000,E1 246.102} C_DIS
LIN {X -0.030,Y -522.656,Z 742.162,A 0.000,B 0.000,C 90.000,E1 245.229} C_DIS
LIN {X 0.005,Y -520.268,Z 742.154,A 0.000,B 0.000,C 90.000,E1 243.768} C_DIS
LIN {X 0.189,Y -518.754,Z 742.149,A 0.000,B 0.000,C 90.000,E1 242.871} C_DIS
LIN {X 0.017,Y -516.539,Z 742.143,A 0.000,B 0.000,C 90.000,E1 241.719} C_DIS
LIN {X 0.060,Y -513.086,Z 742.133,A 0.000,B 0.000,C 90.000,E1 239.950} C_DIS
LIN {X 0.208,Y -510.184,Z 742.125,A 0.000,B 0.000,C 90.000,E1 238.456} C_DIS
LIN {X 0.082,Y -508.403,Z 742.120,A 0.000,B 0.000,C 90.000,E1 237.582} C_DIS
LIN {X -0.066,Y -506.500,Z 742.115,A 0.000,B 0.000,C 90.000,E1 236.707} C_DIS
LIN {X 0.241,Y -503.234,Z 742.107,A 0.000,B 0.000,C 90.000,E1 235.182} C_DIS
LIN {X 0.194,Y -500.406,Z 742.100,A 0.000,B 0.000,C 90.000,E1 233.989} C_DIS
LIN {X -0.297,Y -497.391,Z 742.093,A 0.000,B 0.000,C 90.000,E1 232.844} C_DIS
LIN {X -0.256,Y -492.115,Z 742.082,A 0.000,B 0.000,C 90.000,E1 230.723} C_DIS
LIN {X 0.121,Y -487.816,Z 742.072,A 0.000,B 0.000,C 90.000,E1 228.852} C_DIS
LIN {X -0.053,Y -482.371,Z 742.058,A 0.000,B 0.000,C 90.000,E1 226.419} C_DIS
LIN {X 0.265,Y -479.059,Z 742.049,A 0.000,B 0.000,C 90.000,E1 224.838} C_DIS
LIN {X 0.169,Y -475.815,Z 742.041,A 0.000,B 0.000,C 90.000,E1 223.299} C_DIS
LIN {X 0.121,Y -471.758,Z 742.030,A 0.000,B 0.000,C 90.000,E1 221.434} C_DIS
LIN {X 0.025,Y -467.565,Z 742.020,A 0.000,B 0.000,C 90.000,E1 219.564} C_DIS
LIN {X 0.194,Y -463.473,Z 742.009,A 0.000,B 0.000,C 90.000,E1 217.649} C_DIS
LIN {X 0.201,Y -458.129,Z 741.995,A 0.000,B 0.000,C 90.000,E1 215.105} C_DIS
LIN {X 0.067,Y -453.732,Z 741.983,A 0.000,B 0.000,C 90.000,E1 212.880} C_DIS
LIN {X 0.153,Y -450.724,Z 741.974,A 0.000,B 0.000,C 90.000,E1 211.258} C_DIS
LIN {X 0.095,Y -446.538,Z 741.961,A 0.000,B 0.000,C 90.000,E1 208.999} C_DIS
LIN {X 0.037,Y -442.915,Z 741.950,A 0.000,B 0.000,C 90.000,E1 207.052} C_DIS
LIN {X 0.058,Y -439.829,Z 741.941,A 0.000,B 0.000,C 90.000,E1 205.412} C_DIS
LIN {X -0.137,Y -436.185,Z 741.930,A 0.000,B 0.000,C 90.000,E1 203.462} C_DIS
LIN {X 0.150,Y -433.078,Z 741.921,A 0.000,B 0.000,C 90.000,E1 201.770} C_DIS
LIN {X 0.073,Y -428.709,Z 741.908,A 0.000,B 0.000,C 90.000,E1 199.450} C_DIS
LIN {X 0.154,Y -425.622,Z 741.899,A 0.000,B 0.000,C 90.000,E1 197.764} C_DIS
LIN {X -0.169,Y -421.672,Z 741.888,A 0.000,B 0.000,C 90.000,E1 195.788} C_DIS
LIN {X -0.084,Y -416.642,Z 741.873,A 0.000,B 0.000,C 90.000,E1 193.063} C_DIS
LIN {X -0.151,Y -413.673,Z 741.863,A 0.000,B 0.000,C 90.000,E1 191.366} C_DIS
LIN {X 0.211,Y -408.917,Z 741.848,A 0.000,B 0.000,C 90.000,E1 188.568} C_DIS
LIN {X -0.143,Y -405.577,Z 741.836,A 0.000,B 0.000,C 90.000,E1 186.543} C_DIS
LIN {X 0.084,Y -401.414,Z 741.821,A 0.000,B 0.000,C 90.000,E1 183.726} C_DIS
LIN {X -0.158,Y -398.559,Z 741.809,A 0.000,B 0.000,C 90.000,E1 181.661} C_DIS
LIN {X 0.116,Y -394.884,Z 741.792,A 0.000,B 0.000,C 90.000,E1 178.453} C_DIS
LIN {X 0.116,Y -392.657,Z 741.780,A 0.000,B 0.000,C 90.000,E1 176.331} C_DIS
LIN {X 0.166,Y -389.482,Z 741.758,A 0.000,B 0.000,C 90.000,E1 172.413} C_DIS
LIN {X 0.030,Y -388.066,Z 741.742,A 0.000,B 0.000,C 90.000,E1 169.577} C_DIS
LIN {X -0.131,Y -387.320,Z 741.732,A 0.000,B 0.000,C 90.000,E1 167.813} C_DIS
LIN {X 0.008,Y -386.482,Z 741.720,A 0.000,B 0.000,C 90.000,E1 165.644} C_DIS
LIN {X -0.043,Y -385.807,Z 741.706,A 0.000,B 0.000,C 90.000,E1 163.142} C_DIS
LIN {X 0.121,Y -385.305,Z 741.692,A 0.000,B 0.000,C 90.000,E1 160.604} C_DIS
LIN {X 0.017,Y -384.972,Z 741.680,A 0.000,B 0.000,C 90.000,E1 158.465} C_DIS
LIN {X -0.143,Y -384.642,Z 741.664,A 0.000,B 0.000,C 90.000,E1 155.613} C_DIS
LIN {X -0.028,Y -385.228,Z 741.642,A 0.000,B 0.000,C 90.000,E1 151.641} C_DIS
LIN {X -0.007,Y -386.391,Z 741.629,A 0.000,B 0.000,C 90.000,E1 149.125} C_DIS
LIN {X -0.243,Y -388.425,Z 741.613,A 0.000,B 0.000,C 90.000,E1 146.294} C_DIS
LIN {X 0.072,Y -392.488,Z 741.593,A 0.000,B 0.000,C 90.000,E1 142.683} C_DIS
LIN {X -0.051,Y -395.579,Z 741.583,A 0.000,B 0.000,C 90.000,E1 140.928} C_DIS
LIN {X 0.240,Y -398.242,Z 741.577,A 0.000,B 0.000,C 90.000,E1 139.828} C_DIS
LIN {X -0.230,Y -399.864,Z 741.574,A 0.000,B 0.000,C 90.000,E1 139.380} C_DIS
LIN {X -0.038,Y -403.077,Z 741.570,A 0.000,B 0.000,C 90.000,E1 138.609} C_DIS
LIN {X 0.242,Y -405.430,Z 741.568,A 0.000,B 0.000,C 90.000,E1 138.162} C_DIS
LIN {X 0.077,Y -408.387,Z 741.565,A 0.000,B 0.000,C 90.000,E1 137.757} C_DIS
LIN {X -0.066,Y -414.158,Z 741.562,A 0.000,B 0.000,C 90.000,E1 137.106} C_DIS
LIN {X 0.028,Y -428.585,Z 741.553,A 0.000,B 0.000,C 90.000,E1 135.607} C_DIS
LIN {X 0.098,Y -446.278,Z 741.544,A 0.000,B 0.000,C 90.000,E1 133.866} C_DIS
LIN {X 0.115,Y -454.993,Z 741.539,A 0.000,B 0.000,C 90.000,E1 133.014} C_DIS
LIN {X 0.130,Y -463.501,Z 741.534,A 0.000,B 0.000,C 90.000,E1 132.162} C_DIS
LIN {X 0.100,Y -473.264,Z 741.529,A 0.000,B 0.000,C 90.000,E1 131.148} C_DIS
LIN {X 0.309,Y -478.691,Z 741.525,A 0.000,B 0.000,C 90.000,E1 130.539} C_DIS
LIN {X 0.015,Y -486.789,Z 741.521,A 0.000,B 0.000,C 90.000,E1 129.688} C_DIS
LIN {X 0.304,Y -494.453,Z 741.516,A 0.000,B 0.000,C 90.000,E1 128.749} C_DIS
LIN {X 0.104,Y -500.458,Z 741.511,A 0.000,B 0.000,C 90.000,E1 128.016} C_DIS
LIN {X -0.141,Y -504.936,Z 741.508,A 0.000,B 0.000,C 90.000,E1 127.443} C_DIS
LIN {X 0.051,Y -509.087,Z 741.505,A 0.000,B 0.000,C 90.000,E1 126.824} C_DIS
LIN {X -0.097,Y -515.765,Z 741.499,A 0.000,B 0.000,C 90.000,E1 125.804} C_DIS
LIN {X 0.307,Y -520.160,Z 741.495,A 0.000,B 0.000,C 90.000,E1 125.025} C_DIS
LIN {X 0.077,Y -522.437,Z 741.492,A 0.000,B 0.000,C 90.000,E1 124.612} C_DIS
LIN {X -0.144,Y -524.743,Z 741.490,A 0.000,B 0.000,C 90.000,E1 124.199} C_DIS
LIN {X 0.215,Y -527.627,Z 741.487,A 0.000,B 0.000,C 90.000,E1 123.579} C_DIS
LIN {X -0.027,Y -532.230,Z 741.481,A 0.000,B 0.000,C 90.000,E1 122.594} C_DIS
LIN {X -0.055,Y -536.600,Z 741.476,A 0.000,B 0.000,C 90.000,E1 121.592} C_DIS
LIN {X 0.111,Y -540.130,Z 741.471,A 0.000,B 0.000,C 90.000,E1 120.718} C_DIS
LIN {X 0.038,Y -543.477,Z 741.466,A 0.000,B 0.000,C 90.000,E1 119.873} C_DIS
LIN {X 0.022,Y -547.689,Z 741.460,A 0.000,B 0.000,C 90.000,E1 118.743} C_DIS
LIN {X -0.203,Y -551.554,Z 741.453,A 0.000,B 0.000,C 90.000,E1 117.641} C_DIS
LIN {X 0.119,Y -555.092,Z 741.447,A 0.000,B 0.000,C 90.000,E1 116.488} C_DIS
LIN {X -0.250,Y -557.977,Z 741.441,A 0.000,B 0.000,C 90.000,E1 115.412} C_DIS
LIN {X 0.071,Y -559.280,Z 741.438,A 0.000,B 0.000,C 90.000,E1 114.823} C_DIS
LIN {X -0.044,Y -560.969,Z 741.433,A 0.000,B 0.000,C 90.000,E1 114.003} C_DIS
LIN {X -0.050,Y -562.794,Z 741.427,A 0.000,B 0.000,C 90.000,E1 112.898} C_DIS
LIN {X 0.112,Y -565.176,Z 741.418,A 0.000,B 0.000,C 90.000,E1 111.227} C_DIS
LIN {X 0.120,Y -567.536,Z 741.409,A 0.000,B 0.000,C 90.000,E1 109.577} C_DIS
LIN {X -0.011,Y -569.617,Z 741.400,A 0.000,B 0.000,C 90.000,E1 107.946} C_DIS
LIN {X 0.100,Y -571.244,Z 741.392,A 0.000,B 0.000,C 90.000,E1 106.567} C_DIS
LIN {X 0.236,Y -572.809,Z 741.385,A 0.000,B 0.000,C 90.000,E1 105.190} C_DIS
LIN {X 0.086,Y -574.975,Z 741.374,A 0.000,B 0.000,C 90.000,E1 103.300} C_DIS
LIN {X 0.072,Y -577.492,Z 741.362,A 0.000,B 0.000,C 90.000,E1 101.130} C_DIS
LIN {X 0.137,Y -579.241,Z 741.353,A 0.000,B 0.000,C 90.000,E1 99.500} C_DIS
LIN {X 0.008,Y -580.560,Z 741.345,A 0.000,B 0.000,C 90.000,E1 98.163} C_DIS
LIN {X 0.170,Y -581.633,Z 741.339,A 0.000,B 0.000,C 90.000,E1 97.068} C_DIS
LIN {X -0.005,Y -582.854,Z 741.332,A 0.000,B 0.000,C 90.000,E1 95.739} C_DIS
LIN {X -0.047,Y -584.245,Z 741.323,A 0.000,B 0.000,C 90.000,E1 94.131} C_DIS
LIN {X -0.060,Y -585.490,Z 741.314,A 0.000,B 0.000,C 90.000,E1 92.522} C_DIS
LIN {X -0.274,Y -586.371,Z 741.307,A 0.000,B 0.000,C 90.000,E1 91.203} C_DIS
LIN {X 0.101,Y -587.111,Z 741.299,A 0.000,B 0.000,C 90.000,E1 89.828} C_DIS
LIN {X -0.100,Y -587.657,Z 741.292,A 0.000,B 0.000,C 90.000,E1 88.511} C_DIS
LIN {X -0.279,Y -588.123,Z 741.284,A 0.000,B 0.000,C 90.000,E1 87.192} C_DIS
LIN {X -0.059,Y -588.449,Z 741.278,A 0.000,B 0.000,C 90.000,E1 86.102} C_DIS
LIN {X 0.055,Y -588.716,Z 741.269,A 0.000,B 0.000,C 90.000,E1 84.489} C_DIS
LIN {X 0.186,Y -588.828,Z 741.261,A 0.000,B 0.000,C 90.000,E1 82.875} C_DIS
LIN {X -0.192,Y -588.820,Z 741.252,A 0.000,B 0.000,C 90.000,E1 81.310} C_DIS
LIN {X 0.168,Y -588.676,Z 741.246,A 0.000,B 0.000,C 90.000,E1 80.208} C_DIS
LIN {X -0.117,Y -588.173,Z 741.237,A 0.000,B 0.000,C 90.000,E1 78.634} C_DIS
LIN {X 0.022,Y -587.628,Z 741.229,A 0.000,B 0.000,C 90.000,E1 77.285} C_DIS
LIN {X 0.145,Y -586.988,Z 741.222,A 0.000,B 0.000,C 90.000,E1 75.936} C_DIS
LIN {X 0.070,Y -586.112,Z 741.213,A 0.000,B 0.000,C 90.000,E1 74.338} C_DIS
LIN {X 0.131,Y -585.002,Z 741.204,A 0.000,B 0.000,C 90.000,E1 72.725} C_DIS
LIN {X 0.276,Y -584.199,Z 741.198,A 0.000,B 0.000,C 90.000,E1 71.638} C_DIS
LIN {X 0.066,Y -583.072,Z 741.191,A 0.000,B 0.000,C 90.000,E1 70.315} C_DIS
LIN {X -0.167,Y -582.016,Z 741.185,A 0.000,B 0.000,C 90.000,E1 69.263} C_DIS
LIN {X 0.137,Y -580.953,Z 741.179,A 0.000,B 0.000,C 90.000,E1 68.156} C_DIS
LIN {X -0.115,Y -579.725,Z 741.173,A 0.000,B 0.000,C 90.000,E1 67.102} C_DIS
LIN {X 0.142,Y -578.319,Z 741.167,A 0.000,B 0.000,C 90.000,E1 65.997} C_DIS
LIN {X 0.080,Y -576.796,Z 741.161,A 0.000,B 0.000,C 90.000,E1 64.921} C_DIS
LIN {X -0.003,Y -574.994,Z 741.155,A 0.000,B 0.000,C 90.000,E1 63.845} C_DIS
LIN {X 0.145,Y -572.979,Z 741.149,A 0.000,B 0.000,C 90.000,E1 62.743} C_DIS
LIN {X 0.268,Y -570.697,Z 741.143,A 0.000,B 0.000,C 90.000,E1 61.641} C_DIS
LIN {X 0.033,Y -568.737,Z 741.138,A 0.000,B 0.000,C 90.000,E1 60.845} C_DIS
LIN {X 0.090,Y -565.818,Z 741.132,A 0.000,B 0.000,C 90.000,E1 59.744} C_DIS
LIN {X -0.194,Y -563.417,Z 741.127,A 0.000,B 0.000,C 90.000,E1 58.948} C_DIS
LIN {X -0.208,Y -560.836,Z 741.123,A 0.000,B 0.000,C 90.000,E1 58.122} C_DIS
LIN {X 0.227,Y -557.980,Z 741.118,A 0.000,B 0.000,C 90.000,E1 57.248} C_DIS
LIN {X 0.161,Y -554.824,Z 741.114,A 0.000,B 0.000,C 90.000,E1 56.421} C_DIS
LIN {X -0.126,Y -551.916,Z 741.110,A 0.000,B 0.000,C 90.000,E1 55.754} C_DIS
LIN {X -0.131,Y -548.757,Z 741.106,A 0.000,B 0.000,C 90.000,E1 55.055} C_DIS
LIN {X 0.149,Y -545.220,Z 741.102,A 0.000,B 0.000,C 90.000,E1 54.322} C_DIS
LIN {X 0.082,Y -541.454,Z 741.098,A 0.000,B 0.000,C 90.000,E1 53.623} C_DIS
LIN {X -0.039,Y -539.114,Z 741.096,A 0.000,B 0.000,C 90.000,E1 53.210} C_DIS
LIN {X 0.159,Y -534.641,Z 741.092,A 0.000,B 0.000,C 90.000,E1 52.477} C_DIS
LIN {X 0.157,Y -530.705,Z 741.089,A 0.000,B 0.000,C 90.000,E1 51.904} C_DIS
LIN {X 0.125,Y -526.351,Z 741.085,A 0.000,B 0.000,C 90.000,E1 51.331} C_DIS
LIN {X -0.346,Y -521.405,Z 741.082,A 0.000,B 0.000,C 90.000,E1 50.803} C_DIS
LIN {X -0.204,Y -517.376,Z 741.080,A 0.000,B 0.000,C 90.000,E1 50.356} C_DIS
LIN {X 0.033,Y -511.722,Z 741.077,A 0.000,B 0.000,C 90.000,E1 49.784} C_DIS
LIN {X 0.143,Y -507.294,Z 741.074,A 0.000,B 0.000,C 90.000,E1 49.380} C_DIS
LIN {X -0.271,Y -501.074,Z 741.072,A 0.000,B 0.000,C 90.000,E1 48.933} C_DIS
LIN {X 0.017,Y -493.163,Z 741.069,A 0.000,B 0.000,C 90.000,E1 48.324} C_DIS
LIN {X -0.125,Y -485.119,Z 741.065,A 0.000,B 0.000,C 90.000,E1 47.796} C_DIS
LIN {X -0.001,Y -471.924,Z 741.061,A 0.000,B 0.000,C 90.000,E1 46.944} C_DIS
LIN {X 0.156,Y -449.271,Z 741.053,A 0.000,B 0.000,C 90.000,E1 45.486} C_DIS
LIN {X 0.094,Y -422.103,Z 741.042,A 0.000,B 0.000,C 90.000,E1 43.623} C_DIS
LIN {X -0.069,Y -416.273,Z 741.040,A 0.000,B 0.000,C 90.000,E1 43.176} C_DIS
LIN {X -0.123,Y -414.389,Z 741.039,A 0.000,B 0.000,C 90.000,E1 43.014} C_DIS
LIN {X -0.154,Y -414.352,Z 741.039,A 0.000,B 0.000,C 90.000,E1 43.014} C_DIS
LIN {X 0.061,Y -406.102,Z 741.015,A 0.000,B 0.000,C 90.000,E1 38.624} C_DIS
LIN {X -0.083,Y -403.882,Z 741.009,A 0.000,B 0.000,C 90.000,E1 37.604} C_DIS
LIN {X 0.004,Y -402.957,Z 741.006,A 0.000,B 0.000,C 90.000,E1 37.156} C_DIS
LIN {X 0.182,Y -402.885,Z 741.005,A 0.000,B 0.000,C 90.000,E1 36.870} C_DIS
LIN {X -0.077,Y -403.498,Z 740.986,A 0.000,B 0.000,C 90.000,E1 33.420} C_DIS
LIN {X 0.135,Y -404.852,Z 740.968,A 0.000,B 0.000,C 90.000,E1 30.256} C_DIS
LIN {X 0.146,Y -406.431,Z 740.951,A 0.000,B 0.000,C 90.000,E1 27.129} C_DIS
LIN {X 0.040,Y -408.516,Z 740.934,A 0.000,B 0.000,C 90.000,E1 24.027} C_DIS
LIN {X 0.059,Y -411.219,Z 740.916,A 0.000,B 0.000,C 90.000,E1 20.918} C_DIS
LIN {X 0.122,Y -414.652,Z 740.899,A 0.000,B 0.000,C 90.000,E1 17.819} C_DIS
LIN {X -0.226,Y -418.230,Z 740.884,A 0.000,B 0.000,C 90.000,E1 15.134} C_DIS
LIN {X 0.014,Y -421.242,Z 740.873,A 0.000,B 0.000,C 90.000,E1 13.063} C_DIS
LIN {X 0.222,Y -424.355,Z 740.861,A 0.000,B 0.000,C 90.000,E1 11.007} C_DIS
LIN {X -0.082,Y -427.512,Z 740.850,A 0.000,B 0.000,C 90.000,E1 9.029} C_DIS
LIN {X 0.100,Y -431.162,Z 740.837,A 0.000,B 0.000,C 90.000,E1 6.663} C_DIS
LIN {X 0.030,Y -435.528,Z 740.822,A 0.000,B 0.000,C 90.000,E1 4.012} C_DIS
LIN {X 0.098,Y -438.416,Z 740.813,A 0.000,B 0.000,C 90.000,E1 2.350} C_DIS
LIN {X -0.092,Y -442.132,Z 740.802,A 0.000,B 0.000,C 90.000,E1 0.401} C_DIS
LIN {X 0.093,Y -447.123,Z 740.788,A 0.000,B 0.000,C 90.000,E1 357.822} C_DIS
LIN {X -0.163,Y -451.855,Z 740.775,A 0.000,B 0.000,C 90.000,E1 355.584} C_DIS
LIN {X 0.015,Y -456.199,Z 740.765,A 0.000,B 0.000,C 90.000,E1 353.628} C_DIS
LIN {X -0.114,Y -460.443,Z 740.754,A 0.000,B 0.000,C 90.000,E1 351.724} C_DIS
LIN {X -0.057,Y -463.161,Z 740.747,A 0.000,B 0.000,C 90.000,E1 350.443} C_DIS
LIN {X -0.145,Y -466.279,Z 740.738,A 0.000,B 0.000,C 90.000,E1 348.870} C_DIS
LIN {X 0.004,Y -468.598,Z 740.731,A 0.000,B 0.000,C 90.000,E1 347.589} C_DIS
LIN {X 0.216,Y -471.518,Z 740.722,A 0.000,B 0.000,C 90.000,E1 345.992} C_DIS
LIN {X 0.110,Y -476.325,Z 740.708,A 0.000,B 0.000,C 90.000,E1 343.504} C_DIS
LIN {X -0.119,Y -478.749,Z 740.703,A 0.000,B 0.000,C 90.000,E1 342.598} C_DIS
LIN {X 0.164,Y -480.827,Z 740.700,A 0.000,B 0.000,C 90.000,E1 341.945} C_DIS
LIN {X -0.081,Y -482.973,Z 740.697,A 0.000,B 0.000,C 90.000,E1 341.511} C_DIS
LIN {X -0.009,Y -485.712,Z 740.695,A 0.000,B 0.000,C 90.000,E1 341.040} C_DIS
LIN {X 0.028,Y -488.460,Z 740.693,A 0.000,B 0.000,C 90.000,E1 340.678} C_DIS
LIN {X 0.114,Y -494.534,Z 740.689,A 0.000,B 0.000,C 90.000,E1 340.061} C_DIS
LIN {X -0.107,Y -498.559,Z 740.688,A 0.000,B 0.000,C 90.000,E1 339.752} C_DIS
LIN {X 0.081,Y -506.583,Z 740.684,A 0.000,B 0.000,C 90.000,E1 339.156} C_DIS
LIN {X -0.094,Y -525.683,Z 740.678,A 0.000,B 0.000,C 90.000,E1 337.975} C_DIS
LIN {X 0.158,Y -538.505,Z 740.673,A 0.000,B 0.000,C 90.000,E1 337.177} C_DIS
LIN {X 0.049,Y -541.503,Z 740.672,A 0.000,B 0.000,C 90.000,E1 336.997} C_DIS
LIN {X 0.134,Y -547.525,Z 740.670,A 0.000,B 0.000,C 90.000,E1 336.561} C_DIS
LIN {X 0.190,Y -553.136,Z 740.667,A 0.000,B 0.000,C 90.000,E1 336.102} C_DIS
LIN {X 0.154,Y -558.569,Z 740.665,A 0.000,B 0.000,C 90.000,E1 335.613} C_DIS
LIN {X 0.181,Y -563.812,Z 740.662,A 0.000,B 0.000,C 90.000,E1 335.101} C_DIS
LIN {X 0.067,Y -567.612,Z 740.660,A 0.000,B 0.000,C 90.000,E1 334.717} C_DIS
LIN {X 0.204,Y -573.731,Z 740.656,A 0.000,B 0.000,C 90.000,E1 334.024} C_DIS
LIN {X -0.179,Y -579.683,Z 740.652,A 0.000,B 0.000,C 90.000,E1 333.384} C_DIS
LIN {X -0.009,Y -585.327,Z 740.648,A 0.000,B 0.000,C 90.000,E1 332.692} C_DIS
LIN {X -0.144,Y -592.741,Z 740.643,A 0.000,B 0.000,C 90.000,E1 331.769} C_DIS
LIN {X -0.186,Y -599.734,Z 740.638,A 0.000,B 0.000,C 90.000,E1 330.845} C_DIS
LIN {X -0.140,Y -606.531,Z 740.633,A 0.000,B 0.000,C 90.000,E1 329.921} C_DIS
LIN {X -0.035,Y -613.793,Z 740.627,A 0.000,B 0.000,C 90.000,E1 328.869} C_DIS
LIN {X -0.368,Y -620.575,Z 740.621,A 0.000,B 0.000,C 90.000,E1 327.867} C_DIS
LIN {X -0.281,Y -626.929,Z 740.616,A 0.000,B 0.000,C 90.000,E1 326.834} C_DIS
LIN {X -0.102,Y -632.869,Z 740.610,A 0.000,B 0.000,C 90.000,E1 325.801} C_DIS
LIN {X 0.154,Y -638.421,Z 740.604,A 0.000,B 0.000,C 90.000,E1 324.769} C_DIS
LIN {X -0.070,Y -642.263,Z 740.600,A 0.000,B 0.000,C 90.000,E1 324.036} C_DIS
LIN {X 0.288,Y -646.652,Z 740.595,A 0.000,B 0.000,C 90.000,E1 323.130} C_DIS
LIN {X -0.328,Y -651.312,Z 740.590,A 0.000,B 0.000,C 90.000,E1 322.190} C_DIS
LIN {X 0.029,Y -655.636,Z 740.584,A 0.000,B 0.000,C 90.000,E1 321.170} C_DIS
LIN {X -0.025,Y -658.717,Z 740.580,A 0.000,B 0.000,C 90.000,E1 320.436} C_DIS
LIN {X -0.052,Y -661.661,Z 740.576,A 0.000,B 0.000,C 90.000,E1 319.703} C_DIS
LIN {X 0.381,Y -664.523,Z 740.572,A 0.000,B 0.000,C 90.000,E1 318.933} C_DIS
LIN {X -0.095,Y -667.142,Z 740.568,A 0.000,B 0.000,C 90.000,E1 318.243} C_DIS
LIN {X 0.405,Y -670.471,Z 740.563,A 0.000,B 0.000,C 90.000,E1 317.229} C_DIS
LIN {X 0.019,Y -674.317,Z 740.556,A 0.000,B 0.000,C 90.000,E1 316.053} C_DIS
LIN {X 0.130,Y -677.203,Z 740.551,A 0.000,B 0.000,C 90.000,E1 315.081} C_DIS
LIN {X 0.237,Y -679.209,Z 740.547,A 0.000,B 0.000,C 90.000,E1 314.352} C_DIS
LIN {X 0.086,Y -683.452,Z 740.537,A 0.000,B 0.000,C 90.000,E1 312.690} C_DIS
LIN {X -0.160,Y -685.631,Z 740.532,A 0.000,B 0.000,C 90.000,E1 311.757} C_DIS
LIN {X 0.137,Y -687.707,Z 740.527,A 0.000,B 0.000,C 90.000,E1 310.782} C_DIS
LIN {X -0.065,Y -689.513,Z 740.521,A 0.000,B 0.000,C 90.000,E1 309.850} C_DIS
LIN {X -0.159,Y -691.009,Z 740.516,A 0.000,B 0.000,C 90.000,E1 308.910} C_DIS
LIN {X 0.201,Y -692.343,Z 740.511,A 0.000,B 0.000,C 90.000,E1 307.935} C_DIS
LIN {X 0.087,Y -693.257,Z 740.507,A 0.000,B 0.000,C 90.000,E1 307.237} C_DIS
LIN {X -0.306,Y -694.592,Z 740.500,A 0.000,B 0.000,C 90.000,E1 306.091} C_DIS
LIN {X 0.230,Y -695.497,Z 740.495,A 0.000,B 0.000,C 90.000,E1 305.105} C_DIS
LIN {X 0.430,Y -696.486,Z 740.489,A 0.000,B 0.000,C 90.000,E1 303.913} C_DIS
LIN {X 0.159,Y -697.793,Z 740.479,A 0.000,B 0.000,C 90.000,E1 302.291} C_DIS
LIN {X 0.263,Y -698.912,Z 740.472,A 0.000,B 0.000,C 90.000,E1 300.875} C_DIS
LIN {X -0.159,Y -699.247,Z 740.468,A 0.000,B 0.000,C 90.000,E1 300.207} C_DIS
LIN {X -0.047,Y -699.617,Z 740.461,A 0.000,B 0.000,C 90.000,E1 299.027} C_DIS
LIN {X 0.070,Y -699.975,Z 740.455,A 0.000,B 0.000,C 90.000,E1 297.847} C_DIS
LIN {X 0.140,Y -700.447,Z 740.447,A 0.000,B 0.000,C 90.000,E1 296.437} C_DIS
LIN {X -0.055,Y -701.048,Z 740.440,A 0.000,B 0.000,C 90.000,E1 295.283} C_DIS
LIN {X -0.163,Y -700.959,Z 740.437,A 0.000,B 0.000,C 90.000,E1 294.591} C_DIS
LIN {X 0.382,Y -700.029,Z 740.434,A 0.000,B 0.000,C 90.000,E1 294.079} C_DIS
LIN {X -0.272,Y -699.344,Z 740.433,A 0.000,B 0.000,C 90.000,E1 293.898} C_DIS
LIN {X -0.003,Y -697.835,Z 740.431,A 0.000,B 0.000,C 90.000,E1 293.643} C_DIS
LIN {X 0.384,Y -694.898,Z 740.429,A 0.000,B 0.000,C 90.000,E1 293.259} C_DIS
LIN {X -0.401,Y -693.679,Z 740.429,A 0.000,B 0.000,C 90.000,E1 293.206} C_DIS
LIN {X -0.251,Y -691.809,Z 740.428,A 0.000,B 0.000,C 90.000,E1 293.078} C_DIS
LIN {X -0.382,Y -687.623,Z 740.427,A 0.000,B 0.000,C 90.000,E1 292.898} C_DIS
LIN {X 0.240,Y -685.810,Z 740.427,A 0.000,B 0.000,C 90.000,E1 292.770} C_DIS
LIN {X 0.044,Y -683.851,Z 740.426,A 0.000,B 0.000,C 90.000,E1 292.717} C_DIS
LIN {X -0.018,Y -675.608,Z 740.425,A 0.000,B 0.000,C 90.000,E1 292.514} C_DIS
LIN {X 0.060,Y -666.678,Z 740.424,A 0.000,B 0.000,C 90.000,E1 292.386} C_DIS
LIN {X -0.099,Y -660.519,Z 740.424,A 0.000,B 0.000,C 90.000,E1 292.333} C_DIS
LIN {X -0.328,Y -647.246,Z 740.423,A 0.000,B 0.000,C 90.000,E1 292.153} C_DIS
LIN {X -0.237,Y -634.400,Z 740.422,A 0.000,B 0.000,C 90.000,E1 291.897} C_DIS
LIN {X -0.217,Y -621.162,Z 740.420,A 0.000,B 0.000,C 90.000,E1 291.589} C_DIS
LIN {X 0.179,Y -604.050,Z 740.417,A 0.000,B 0.000,C 90.000,E1 291.099} C_DIS
LIN {X 0.122,Y -576.016,Z 740.413,A 0.000,B 0.000,C 90.000,E1 290.301} C_DIS
LIN {X 0.014,Y -568.660,Z 740.412,A 0.000,B 0.000,C 90.000,E1 290.120} C_DIS
LIN {X 0.062,Y -563.213,Z 740.411,A 0.000,B 0.000,C 90.000,E1 289.939} C_DIS
LIN {X 0.014,Y -561.579,Z 740.411,A 0.000,B 0.000,C 90.000,E1 289.885} C_DIS
LIN {X 0.307,Y -557.405,Z 740.409,A 0.000,B 0.000,C 90.000,E1 289.631} C_DIS
LIN {X -0.016,Y -556.840,Z 740.409,A 0.000,B 0.000,C 90.000,E1 289.631} C_DIS
LIN {X -0.070,Y -556.779,Z 740.409,A 0.000,B 0.000,C 90.000,E1 289.631} C_DIS
LIN {X -0.146,Y -555.610,Z 740.408,A 0.000,B 0.000,C 90.000,E1 289.450} C_DIS
LIN {X -0.156,Y -554.912,Z 740.406,A 0.000,B 0.000,C 90.000,E1 289.033} C_DIS
LIN {X -0.262,Y -554.349,Z 740.397,A 0.000,B 0.000,C 90.000,E1 287.457} C_DIS
LIN {X 0.097,Y -553.798,Z 740.389,A 0.000,B 0.000,C 90.000,E1 286.024} C_DIS
LIN {X 0.146,Y -553.116,Z 740.378,A 0.000,B 0.000,C 90.000,E1 284.064} C_DIS
LIN {X 0.034,Y -552.511,Z 740.367,A 0.000,B 0.000,C 90.000,E1 282.119} C_DIS
LIN {X 0.104,Y -551.937,Z 740.358,A 0.000,B 0.000,C 90.000,E1 280.433} C_DIS
LIN {X 0.142,Y -551.304,Z 740.350,A 0.000,B 0.000,C 90.000,E1 279.029} C_DIS
LIN {X 0.136,Y -550.366,Z 740.339,A 0.000,B 0.000,C 90.000,E1 277.068} C_DIS
LIN {X 0.114,Y -549.474,Z 740.328,A 0.000,B 0.000,C 90.000,E1 275.106} C_DIS
LIN {X -0.123,Y -548.807,Z 740.321,A 0.000,B 0.000,C 90.000,E1 273.726} C_DIS
LIN {X 0.258,Y -547.793,Z 740.310,A 0.000,B 0.000,C 90.000,E1 271.718} C_DIS
LIN {X -0.150,Y -547.419,Z 740.305,A 0.000,B 0.000,C 90.000,E1 270.917} C_DIS
LIN {X 0.123,Y -546.385,Z 740.296,A 0.000,B 0.000,C 90.000,E1 269.198} C_DIS
LIN {X -0.163,Y -545.275,Z 740.286,A 0.000,B 0.000,C 90.000,E1 267.535} C_DIS
LIN {X 0.104,Y -544.226,Z 740.277,A 0.000,B 0.000,C 90.000,E1 265.812} C_DIS
LIN {X -0.219,Y -543.249,Z 740.269,A 0.000,B 0.000,C 90.000,E1 264.432} C_DIS
LIN {X -0.030,Y -542.188,Z 740.261,A 0.000,B 0.000,C 90.000,E1 262.996} C_DIS
LIN {X 0.270,Y -541.087,Z 740.253,A 0.000,B 0.000,C 90.000,E1 261.546} C_DIS
LIN {X 0.097,Y -539.649,Z 740.244,A 0.000,B 0.000,C 90.000,E1 259.859} C_DIS
LIN {X -0.045,Y -538.025,Z 740.233,A 0.000,B 0.000,C 90.000,E1 257.881} C_DIS
LIN {X -0.193,Y -537.053,Z 740.226,A 0.000,B 0.000,C 90.000,E1 256.756} C_DIS
LIN {X 0.043,Y -535.981,Z 740.220,A 0.000,B 0.000,C 90.000,E1 255.589} C_DIS
LIN {X 0.099,Y -534.145,Z 740.210,A 0.000,B 0.000,C 90.000,E1 253.866} C_DIS
LIN {X -0.240,Y -532.296,Z 740.201,A 0.000,B 0.000,C 90.000,E1 252.181} C_DIS
LIN {X -0.317,Y -531.011,Z 740.195,A 0.000,B 0.000,C 90.000,E1 251.040} C_DIS
LIN {X -0.056,Y -529.063,Z 740.187,A 0.000,B 0.000,C 90.000,E1 249.571} C_DIS
LIN {X 0.169,Y -527.134,Z 740.179,A 0.000,B 0.000,C 90.000,E1 248.103} C_DIS
LIN {X 0.235,Y -524.539,Z 740.169,A 0.000,B 0.000,C 90.000,E1 246.357} C_DIS
LIN {X -0.072,Y -522.716,Z 740.162,A 0.000,B 0.000,C 90.000,E1 245.229} C_DIS
LIN {X -0.036,Y -520.320,Z 740.154,A 0.000,B 0.000,C 90.000,E1 243.768} C_DIS
LIN {X 0.148,Y -518.803,Z 740.149,A 0.000,B 0.000,C 90.000,E1 242.871} C_DIS
LIN {X -0.022,Y -516.588,Z 740.143,A 0.000,B 0.000,C 90.000,E1 241.719} C_DIS
LIN {X -0.076,Y -513.695,Z 740.135,A 0.000,B 0.000,C 90.000,E1 240.255} C_DIS
LIN {X 0.170,Y -510.207,Z 740.125,A 0.000,B 0.000,C 90.000,E1 238.456} C_DIS
LIN {X 0.045,Y -508.429,Z 740.120,A 0.000,B 0.000,C 90.000,E1 237.582} C_DIS
LIN {X -0.103,Y -506.528,Z 740.115,A 0.000,B 0.000,C 90.000,E1 236.707} C_DIS
LIN {X 0.205,Y -503.265,Z 740.107,A 0.000,B 0.000,C 90.000,E1 235.182} C_DIS
LIN {X 0.158,Y -500.415,Z 740.100,A 0.000,B 0.000,C 90.000,E1 233.989} C_DIS
LIN {X 0.064,Y -497.415,Z 740.093,A 0.000,B 0.000,C 90.000,E1 232.798} C_DIS
LIN {X 0.090,Y -492.150,Z 740.082,A 0.000,B 0.000,C 90.000,E1 230.678} C_DIS
LIN {X 0.087,Y -487.855,Z 740.072,A 0.000,B 0.000,C 90.000,E1 228.852} C_DIS
LIN {X -0.282,Y -481.744,Z 740.056,A 0.000,B 0.000,C 90.000,E1 226.134} C_DIS
LIN {X -0.085,Y -477.082,Z 740.044,A 0.000,B 0.000,C 90.000,E1 223.947} C_DIS
LIN {X 0.025,Y -474.468,Z 740.037,A 0.000,B 0.000,C 90.000,E1 222.690} C_DIS
LIN {X 0.090,Y -471.785,Z 740.030,A 0.000,B 0.000,C 90.000,E1 221.434} C_DIS
LIN {X -0.073,Y -468.292,Z 740.022,A 0.000,B 0.000,C 90.000,E1 219.886} C_DIS
LIN {X 0.165,Y -463.482,Z 740.009,A 0.000,B 0.000,C 90.000,E1 217.649} C_DIS
LIN {X 0.060,Y -458.785,Z 739.997,A 0.000,B 0.000,C 90.000,E1 215.438} C_DIS
LIN {X 0.038,Y -453.776,Z 739.983,A 0.000,B 0.000,C 90.000,E1 212.880} C_DIS
LIN {X 0.126,Y -450.732,Z 739.974,A 0.000,B 0.000,C 90.000,E1 211.258} C_DIS
LIN {X -0.003,Y -447.130,Z 739.963,A 0.000,B 0.000,C 90.000,E1 209.333} C_DIS
LIN {X -0.099,Y -444.154,Z 739.954,A 0.000,B 0.000,C 90.000,E1 207.719} C_DIS
LIN {X 0.186,Y -440.464,Z 739.943,A 0.000,B 0.000,C 90.000,E1 205.720} C_DIS
LIN {X -0.163,Y -436.230,Z 739.930,A 0.000,B 0.000,C 90.000,E1 203.462} C_DIS
LIN {X 0.126,Y -433.100,Z 739.921,A 0.000,B 0.000,C 90.000,E1 201.770} C_DIS
LIN {X 0.049,Y -428.753,Z 739.908,A 0.000,B 0.000,C 90.000,E1 199.450} C_DIS
LIN {X 0.131,Y -425.660,Z 739.899,A 0.000,B 0.000,C 90.000,E1 197.764} C_DIS
LIN {X 0.151,Y -422.394,Z 739.889,A 0.000,B 0.000,C 90.000,E1 196.079} C_DIS
LIN {X -0.157,Y -417.325,Z 739.874,A 0.000,B 0.000,C 90.000,E1 193.411} C_DIS
LIN {X -0.169,Y -413.777,Z 739.863,A 0.000,B 0.000,C 90.000,E1 191.366} C_DIS
LIN {X 0.196,Y -408.984,Z 739.848,A 0.000,B 0.000,C 90.000,E1 188.568} C_DIS
LIN {X -0.166,Y -406.224,Z 739.838,A 0.000,B 0.000,C 90.000,E1 186.891} C_DIS
LIN {X 0.075,Y -401.500,Z 739.821,A 0.000,B 0.000,C 90.000,E1 183.726} C_DIS
LIN {X -0.165,Y -398.650,Z 739.809,A 0.000,B 0.000,C 90.000,E1 181.661} C_DIS
LIN {X 0.178,Y -395.377,Z 739.794,A 0.000,B 0.000,C 90.000,E1 178.797} C_DIS
LIN {X -0.147,Y -393.546,Z 739.784,A 0.000,B 0.000,C 90.000,E1 177.078} C_DIS
LIN {X -0.052,Y -390.330,Z 739.764,A 0.000,B 0.000,C 90.000,E1 173.514} C_DIS
LIN {X 0.009,Y -389.170,Z 739.754,A 0.000,B 0.000,C 90.000,E1 171.724} C_DIS
LIN {X 0.053,Y -388.100,Z 739.740,A 0.000,B 0.000,C 90.000,E1 169.218} C_DIS
LIN {X -0.115,Y -387.498,Z 739.732,A 0.000,B 0.000,C 90.000,E1 167.813} C_DIS
LIN {X 0.029,Y -386.695,Z 739.720,A 0.000,B 0.000,C 90.000,E1 165.644} C_DIS
LIN {X -0.016,Y -386.018,Z 739.706,A 0.000,B 0.000,C 90.000,E1 163.142} C_DIS
LIN {X 0.155,Y -385.595,Z 739.692,A 0.000,B 0.000,C 90.000,E1 160.604} C_DIS
LIN {X -0.101,Y -385.300,Z 739.682,A 0.000,B 0.000,C 90.000,E1 158.847} C_DIS
LIN {X 0.085,Y -384.958,Z 739.668,A 0.000,B 0.000,C 90.000,E1 156.305} C_DIS
LIN {X 0.046,Y -385.106,Z 739.651,A 0.000,B 0.000,C 90.000,E1 153.076} C_DIS
LIN {X 0.062,Y -386.608,Z 739.629,A 0.000,B 0.000,C 90.000,E1 149.125} C_DIS
LIN {X -0.166,Y -388.569,Z 739.613,A 0.000,B 0.000,C 90.000,E1 146.294} C_DIS
LIN {X -0.085,Y -392.507,Z 739.593,A 0.000,B 0.000,C 90.000,E1 142.718} C_DIS
LIN {X 0.031,Y -395.468,Z 739.583,A 0.000,B 0.000,C 90.000,E1 140.928} C_DIS
LIN {X -0.240,Y -397.981,Z 739.577,A 0.000,B 0.000,C 90.000,E1 139.908} C_DIS
LIN {X -0.156,Y -399.481,Z 739.574,A 0.000,B 0.000,C 90.000,E1 139.380} C_DIS
LIN {X 0.018,Y -402.379,Z 739.570,A 0.000,B 0.000,C 90.000,E1 138.609} C_DIS
LIN {X 0.033,Y -404.445,Z 739.568,A 0.000,B 0.000,C 90.000,E1 138.243} C_DIS
LIN {X -0.057,Y -405.316,Z 739.567,A 0.000,B 0.000,C 90.000,E1 138.081} C_DIS
LIN {X -0.009,Y -408.849,Z 739.564,A 0.000,B 0.000,C 90.000,E1 137.553} C_DIS
LIN {X -0.178,Y -413.189,Z 739.561,A 0.000,B 0.000,C 90.000,E1 137.067} C_DIS
LIN {X -0.150,Y -427.739,Z 739.553,A 0.000,B 0.000,C 90.000,E1 135.567} C_DIS
LIN {X -0.227,Y -446.952,Z 739.543,A 0.000,B 0.000,C 90.000,E1 133.704} C_DIS
LIN {X -0.009,Y -454.213,Z 739.539,A 0.000,B 0.000,C 90.000,E1 132.975} C_DIS
LIN {X -0.137,Y -464.159,Z 739.533,A 0.000,B 0.000,C 90.000,E1 132.000} C_DIS
LIN {X -0.123,Y -473.918,Z 739.528,A 0.000,B 0.000,C 90.000,E1 130.987} C_DIS
LIN {X -0.138,Y -480.773,Z 739.524,A 0.000,B 0.000,C 90.000,E1 130.253} C_DIS
LIN {X 0.133,Y -487.490,Z 739.519,A 0.000,B 0.000,C 90.000,E1 129.483} C_DIS
LIN {X 0.112,Y -495.222,Z 739.515,A 0.000,B 0.000,C 90.000,E1 128.588} C_DIS
LIN {X 0.208,Y -499.751,Z 739.511,A 0.000,B 0.000,C 90.000,E1 128.016} C_DIS
LIN {X 0.093,Y -504.213,Z 739.508,A 0.000,B 0.000,C 90.000,E1 127.443} C_DIS
LIN {X 0.029,Y -508.357,Z 739.505,A 0.000,B 0.000,C 90.000,E1 126.870} C_DIS
LIN {X -0.051,Y -513.219,Z 739.501,A 0.000,B 0.000,C 90.000,E1 126.137} C_DIS
LIN {X 0.095,Y -516.098,Z 739.498,A 0.000,B 0.000,C 90.000,E1 125.678} C_DIS
LIN {X -0.039,Y -519.609,Z 739.495,A 0.000,B 0.000,C 90.000,E1 125.105} C_DIS
LIN {X 0.232,Y -524.320,Z 739.490,A 0.000,B 0.000,C 90.000,E1 124.199} C_DIS
LIN {X -0.012,Y -527.919,Z 739.486,A 0.000,B 0.000,C 90.000,E1 123.499} C_DIS
LIN {X 0.061,Y -531.903,Z 739.481,A 0.000,B 0.000,C 90.000,E1 122.625} C_DIS
LIN {X -0.273,Y -535.665,Z 739.477,A 0.000,B 0.000,C 90.000,E1 121.799} C_DIS
LIN {X -0.257,Y -539.872,Z 739.471,A 0.000,B 0.000,C 90.000,E1 120.797} C_DIS
LIN {X -0.060,Y -543.253,Z 739.466,A 0.000,B 0.000,C 90.000,E1 119.922} C_DIS
LIN {X 0.147,Y -548.533,Z 739.458,A 0.000,B 0.000,C 90.000,E1 118.487} C_DIS
LIN {X -0.064,Y -552.348,Z 739.452,A 0.000,B 0.000,C 90.000,E1 117.385} C_DIS
LIN {X -0.004,Y -554.996,Z 739.448,A 0.000,B 0.000,C 90.000,E1 116.539} C_DIS
LIN {X 0.124,Y -557.934,Z 739.441,A 0.000,B 0.000,C 90.000,E1 115.412} C_DIS
LIN {X -0.297,Y -559.291,Z 739.438,A 0.000,B 0.000,C 90.000,E1 114.899} C_DIS
LIN {X 0.103,Y -561.033,Z 739.434,A 0.000,B 0.000,C 90.000,E1 114.027} C_DIS
LIN {X -0.190,Y -562.866,Z 739.427,A 0.000,B 0.000,C 90.000,E1 112.950} C_DIS
LIN {X -0.162,Y -564.486,Z 739.421,A 0.000,B 0.000,C 90.000,E1 111.844} C_DIS
LIN {X 0.228,Y -566.484,Z 739.414,A 0.000,B 0.000,C 90.000,E1 110.429} C_DIS
LIN {X 0.119,Y -568.057,Z 739.408,A 0.000,B 0.000,C 90.000,E1 109.341} C_DIS
LIN {X 0.179,Y -570.154,Z 739.398,A 0.000,B 0.000,C 90.000,E1 107.692} C_DIS
LIN {X -0.051,Y -571.470,Z 739.392,A 0.000,B 0.000,C 90.000,E1 106.622} C_DIS
LIN {X -0.279,Y -573.412,Z 739.383,A 0.000,B 0.000,C 90.000,E1 105.009} C_DIS
LIN {X -0.064,Y -575.268,Z 739.374,A 0.000,B 0.000,C 90.000,E1 103.355} C_DIS
LIN {X -0.075,Y -577.823,Z 739.362,A 0.000,B 0.000,C 90.000,E1 101.186} C_DIS
LIN {X -0.006,Y -579.602,Z 739.353,A 0.000,B 0.000,C 90.000,E1 99.557} C_DIS
LIN {X -0.130,Y -580.942,Z 739.346,A 0.000,B 0.000,C 90.000,E1 98.219} C_DIS
LIN {X 0.033,Y -582.022,Z 739.340,A 0.000,B 0.000,C 90.000,E1 97.125} C_DIS
LIN {X 0.030,Y -583.501,Z 739.331,A 0.000,B 0.000,C 90.000,E1 95.511} C_DIS
LIN {X -0.171,Y -584.688,Z 739.323,A 0.000,B 0.000,C 90.000,E1 94.188} C_DIS
LIN {X -0.177,Y -585.951,Z 739.314,A 0.000,B 0.000,C 90.000,E1 92.579} C_DIS
LIN {X 0.204,Y -586.839,Z 739.307,A 0.000,B 0.000,C 90.000,E1 91.203} C_DIS
LIN {X 0.001,Y -587.603,Z 739.299,A 0.000,B 0.000,C 90.000,E1 89.885} C_DIS
LIN {X -0.191,Y -588.167,Z 739.292,A 0.000,B 0.000,C 90.000,E1 88.568} C_DIS
LIN {X -0.167,Y -588.738,Z 739.283,A 0.000,B 0.000,C 90.000,E1 86.963} C_DIS
LIN {X 0.102,Y -589.009,Z 739.277,A 0.000,B 0.000,C 90.000,E1 85.869} C_DIS
LIN {X -0.008,Y -589.217,Z 739.270,A 0.000,B 0.000,C 90.000,E1 84.546} C_DIS
LIN {X 0.135,Y -589.331,Z 739.261,A 0.000,B 0.000,C 90.000,E1 82.932} C_DIS
LIN {X -0.319,Y -589.299,Z 739.252,A 0.000,B 0.000,C 90.000,E1 81.376} C_DIS
LIN {X 0.039,Y -589.158,Z 739.246,A 0.000,B 0.000,C 90.000,E1 80.274} C_DIS
LIN {X -0.078,Y -588.804,Z 739.240,A 0.000,B 0.000,C 90.000,E1 79.218} C_DIS
LIN {X -0.309,Y -588.431,Z 739.234,A 0.000,B 0.000,C 90.000,E1 78.173} C_DIS
LIN {X 0.077,Y -587.686,Z 739.225,A 0.000,B 0.000,C 90.000,E1 76.533} C_DIS
LIN {X 0.083,Y -587.085,Z 739.219,A 0.000,B 0.000,C 90.000,E1 75.463} C_DIS
LIN {X -0.235,Y -586.319,Z 739.212,A 0.000,B 0.000,C 90.000,E1 74.157} C_DIS
LIN {X -0.166,Y -585.171,Z 739.203,A 0.000,B 0.000,C 90.000,E1 72.543} C_DIS
LIN {X -0.019,Y -584.309,Z 739.197,A 0.000,B 0.000,C 90.000,E1 71.456} C_DIS
LIN {X -0.028,Y -583.147,Z 739.190,A 0.000,B 0.000,C 90.000,E1 70.115} C_DIS
LIN {X 0.343,Y -581.527,Z 739.181,A 0.000,B 0.000,C 90.000,E1 68.465} C_DIS
LIN {X 0.099,Y -580.318,Z 739.175,A 0.000,B 0.000,C 90.000,E1 67.411} C_DIS
LIN {X -0.162,Y -578.940,Z 739.169,A 0.000,B 0.000,C 90.000,E1 66.357} C_DIS
LIN {X 0.169,Y -577.011,Z 739.161,A 0.000,B 0.000,C 90.000,E1 64.973} C_DIS
LIN {X 0.094,Y -575.163,Z 739.155,A 0.000,B 0.000,C 90.000,E1 63.896} C_DIS
LIN {X 0.145,Y -573.646,Z 739.151,A 0.000,B 0.000,C 90.000,E1 63.076} C_DIS
LIN {X 0.091,Y -572.592,Z 739.148,A 0.000,B 0.000,C 90.000,E1 62.538} C_DIS
LIN {X 0.108,Y -570.789,Z 739.143,A 0.000,B 0.000,C 90.000,E1 61.719} C_DIS
LIN {X -0.129,Y -568.804,Z 739.138,A 0.000,B 0.000,C 90.000,E1 60.923} C_DIS
LIN {X 0.210,Y -565.861,Z 739.132,A 0.000,B 0.000,C 90.000,E1 59.793} C_DIS
LIN {X -0.070,Y -563.416,Z 739.128,A 0.000,B 0.000,C 90.000,E1 58.997} C_DIS
LIN {X 0.100,Y -560.794,Z 739.123,A 0.000,B 0.000,C 90.000,E1 58.152} C_DIS
LIN {X 0.057,Y -557.921,Z 739.119,A 0.000,B 0.000,C 90.000,E1 57.327} C_DIS
LIN {X -0.012,Y -554.712,Z 739.114,A 0.000,B 0.000,C 90.000,E1 56.501} C_DIS
LIN {X 0.009,Y -551.757,Z 739.110,A 0.000,B 0.000,C 90.000,E1 55.801} C_DIS
LIN {X 0.004,Y -548.538,Z 739.106,A 0.000,B 0.000,C 90.000,E1 55.102} C_DIS
LIN {X -0.033,Y -544.960,Z 739.102,A 0.000,B 0.000,C 90.000,E1 54.402} C_DIS
LIN {X -0.102,Y -541.094,Z 739.098,A 0.000,B 0.000,C 90.000,E1 53.703} C_DIS
LIN {X 0.096,Y -538.719,Z 739.096,A 0.000,B 0.000,C 90.000,E1 53.256} C_DIS
LIN {X -0.032,Y -534.194,Z 739.092,A 0.000,B 0.000,C 90.000,E1 52.557} C_DIS
LIN {X 0.095,Y -530.284,Z 739.089,A 0.000,B 0.000,C 90.000,E1 51.984} C_DIS
LIN {X -0.141,Y -526.046,Z 739.086,A 0.000,B 0.000,C 90.000,E1 51.457} C_DIS
LIN {X -0.206,Y -520.974,Z 739.083,A 0.000,B 0.000,C 90.000,E1 50.884} C_DIS
LIN {X -0.031,Y -516.942,Z 739.080,A 0.000,B 0.000,C 90.000,E1 50.436} C_DIS
LIN {X -0.104,Y -511.280,Z 739.077,A 0.000,B 0.000,C 90.000,E1 49.908} C_DIS
LIN {X -0.129,Y -507.057,Z 739.075,A 0.000,B 0.000,C 90.000,E1 49.542} C_DIS
LIN {X 0.184,Y -500.806,Z 739.072,A 0.000,B 0.000,C 90.000,E1 49.013} C_DIS
LIN {X 0.031,Y -494.388,Z 739.070,A 0.000,B 0.000,C 90.000,E1 48.566} C_DIS
LIN {X -0.033,Y -489.658,Z 739.068,A 0.000,B 0.000,C 90.000,E1 48.243} C_DIS
LIN {X -0.038,Y -481.411,Z 739.065,A 0.000,B 0.000,C 90.000,E1 47.715} C_DIS
LIN {X 0.213,Y -471.660,Z 739.062,A 0.000,B 0.000,C 90.000,E1 47.067} C_DIS
LIN {X 0.026,Y -445.858,Z 739.053,A 0.000,B 0.000,C 90.000,E1 45.445} C_DIS
LIN {X -0.274,Y -423.428,Z 739.044,A 0.000,B 0.000,C 90.000,E1 43.947} C_DIS
LIN {X -0.011,Y -415.810,Z 739.041,A 0.000,B 0.000,C 90.000,E1 43.299} C_DIS
LIN {X -0.055,Y -414.838,Z 739.040,A 0.000,B 0.000,C 90.000,E1 43.218} C_DIS
LIN {X -0.084,Y -414.827,Z 739.040,A 0.000,B 0.000,C 90.000,E1 43.218} C_DIS
LIN {X -0.046,Y -406.207,Z 739.015,A 0.000,B 0.000,C 90.000,E1 38.705} C_DIS
LIN {X 0.099,Y -405.568,Z 739.013,A 0.000,B 0.000,C 90.000,E1 38.338} C_DIS
LIN {X -0.051,Y -403.279,Z 739.007,A 0.000,B 0.000,C 90.000,E1 37.317} C_DIS
LIN {X 0.082,Y -403.204,Z 739.005,A 0.000,B 0.000,C 90.000,E1 36.950} C_DIS
LIN {X -0.159,Y -403.840,Z 738.986,A 0.000,B 0.000,C 90.000,E1 33.499} C_DIS
LIN {X 0.073,Y -405.192,Z 738.969,A 0.000,B 0.000,C 90.000,E1 30.335} C_DIS
LIN {X 0.121,Y -406.379,Z 738.955,A 0.000,B 0.000,C 90.000,E1 27.897} C_DIS
LIN {X 0.180,Y -407.842,Z 738.942,A 0.000,B 0.000,C 90.000,E1 25.463} C_DIS
LIN {X -0.076,Y -409.125,Z 738.932,A 0.000,B 0.000,C 90.000,E1 23.770} C_DIS
LIN {X -0.042,Y -411.919,Z 738.915,A 0.000,B 0.000,C 90.000,E1 20.663} C_DIS
LIN {X -0.093,Y -415.400,Z 738.898,A 0.000,B 0.000,C 90.000,E1 17.583} C_DIS
LIN {X 0.097,Y -418.994,Z 738.883,A 0.000,B 0.000,C 90.000,E1 14.828} C_DIS
LIN {X 0.184,Y -421.508,Z 738.873,A 0.000,B 0.000,C 90.000,E1 13.119} C_DIS
LIN {X -0.101,Y -424.591,Z 738.862,A 0.000,B 0.000,C 90.000,E1 11.130} C_DIS
LIN {X 0.031,Y -427.724,Z 738.851,A 0.000,B 0.000,C 90.000,E1 9.095} C_DIS
LIN {X 0.173,Y -430.852,Z 738.839,A 0.000,B 0.000,C 90.000,E1 7.068} C_DIS
LIN {X 0.102,Y -435.129,Z 738.825,A 0.000,B 0.000,C 90.000,E1 4.416} C_DIS
LIN {X -0.147,Y -438.547,Z 738.814,A 0.000,B 0.000,C 90.000,E1 2.465} C_DIS
LIN {X 0.106,Y -442.248,Z 738.803,A 0.000,B 0.000,C 90.000,E1 0.458} C_DIS
LIN {X 0.100,Y -447.371,Z 738.788,A 0.000,B 0.000,C 90.000,E1 357.822} C_DIS
LIN {X -0.150,Y -452.068,Z 738.775,A 0.000,B 0.000,C 90.000,E1 355.584} C_DIS
LIN {X 0.034,Y -456.404,Z 738.765,A 0.000,B 0.000,C 90.000,E1 353.628} C_DIS
LIN {X -0.092,Y -460.618,Z 738.754,A 0.000,B 0.000,C 90.000,E1 351.724} C_DIS
LIN {X -0.030,Y -463.329,Z 738.747,A 0.000,B 0.000,C 90.000,E1 350.443} C_DIS
LIN {X -0.117,Y -466.439,Z 738.738,A 0.000,B 0.000,C 90.000,E1 348.870} C_DIS
LIN {X 0.035,Y -468.762,Z 738.731,A 0.000,B 0.000,C 90.000,E1 347.589} C_DIS
LIN {X 0.251,Y -471.677,Z 738.722,A 0.000,B 0.000,C 90.000,E1 345.992} C_DIS
LIN {X 0.117,Y -477.105,Z 738.707,A 0.000,B 0.000,C 90.000,E1 343.196} C_DIS
LIN {X -0.246,Y -479.515,Z 738.702,A 0.000,B 0.000,C 90.000,E1 342.308} C_DIS
LIN {X 0.179,Y -481.682,Z 738.698,A 0.000,B 0.000,C 90.000,E1 341.638} C_DIS
LIN {X 0.058,Y -483.413,Z 738.696,A 0.000,B 0.000,C 90.000,E1 341.275} C_DIS
LIN {X -0.109,Y -485.614,Z 738.694,A 0.000,B 0.000,C 90.000,E1 340.913} C_DIS
LIN {X 0.136,Y -489.014,Z 738.691,A 0.000,B 0.000,C 90.000,E1 340.423} C_DIS
LIN {X 0.209,Y -493.559,Z 738.689,A 0.000,B 0.000,C 90.000,E1 339.934} C_DIS
LIN {X -0.003,Y -499.827,Z 738.686,A 0.000,B 0.000,C 90.000,E1 339.444} C_DIS
LIN {X -0.096,Y -507.650,Z 738.683,A 0.000,B 0.000,C 90.000,E1 338.901} C_DIS
LIN {X -0.213,Y -535.039,Z 738.673,A 0.000,B 0.000,C 90.000,E1 337.230} C_DIS
LIN {X 0.001,Y -539.692,Z 738.672,A 0.000,B 0.000,C 90.000,E1 336.922} C_DIS
LIN {X 0.151,Y -545.747,Z 738.669,A 0.000,B 0.000,C 90.000,E1 336.485} C_DIS
LIN {X -0.001,Y -551.525,Z 738.667,A 0.000,B 0.000,C 90.000,E1 336.049} C_DIS
LIN {X 0.290,Y -556.964,Z 738.664,A 0.000,B 0.000,C 90.000,E1 335.537} C_DIS
LIN {X 0.124,Y -562.267,Z 738.661,A 0.000,B 0.000,C 90.000,E1 335.049} C_DIS
LIN {X 0.016,Y -567.384,Z 738.659,A 0.000,B 0.000,C 90.000,E1 334.537} C_DIS
LIN {X 0.060,Y -574.787,Z 738.654,A 0.000,B 0.000,C 90.000,E1 333.717} C_DIS
LIN {X -0.195,Y -583.010,Z 738.649,A 0.000,B 0.000,C 90.000,E1 332.794} C_DIS
LIN {X -0.055,Y -589.507,Z 738.644,A 0.000,B 0.000,C 90.000,E1 331.975} C_DIS
LIN {X -0.090,Y -595.725,Z 738.640,A 0.000,B 0.000,C 90.000,E1 331.179} C_DIS
LIN {X -0.166,Y -604.583,Z 738.633,A 0.000,B 0.000,C 90.000,E1 329.999} C_DIS
LIN {X -0.014,Y -609.276,Z 738.630,A 0.000,B 0.000,C 90.000,E1 329.331} C_DIS
LIN {X 0.162,Y -614.647,Z 738.625,A 0.000,B 0.000,C 90.000,E1 328.535} C_DIS
LIN {X -0.148,Y -620.596,Z 738.620,A 0.000,B 0.000,C 90.000,E1 327.661} C_DIS
LIN {X -0.051,Y -626.208,Z 738.615,A 0.000,B 0.000,C 90.000,E1 326.755} C_DIS
LIN {X 0.125,Y -632.933,Z 738.609,A 0.000,B 0.000,C 90.000,E1 325.595} C_DIS
LIN {X -0.138,Y -638.457,Z 738.603,A 0.000,B 0.000,C 90.000,E1 324.609} C_DIS
LIN {X -0.316,Y -644.274,Z 738.597,A 0.000,B 0.000,C 90.000,E1 323.497} C_DIS
LIN {X 0.018,Y -647.347,Z 738.594,A 0.000,B 0.000,C 90.000,E1 322.844} C_DIS
LIN {X -0.114,Y -650.844,Z 738.589,A 0.000,B 0.000,C 90.000,E1 322.110} C_DIS
LIN {X 0.240,Y -655.268,Z 738.584,A 0.000,B 0.000,C 90.000,E1 321.090} C_DIS
LIN {X 0.145,Y -659.393,Z 738.579,A 0.000,B 0.000,C 90.000,E1 320.114} C_DIS
LIN {X 0.105,Y -663.304,Z 738.573,A 0.000,B 0.000,C 90.000,E1 319.138} C_DIS
LIN {X 0.120,Y -666.101,Z 738.569,A 0.000,B 0.000,C 90.000,E1 318.405} C_DIS
